Yaskawa INFORM job: test_long_tjr1.JBI

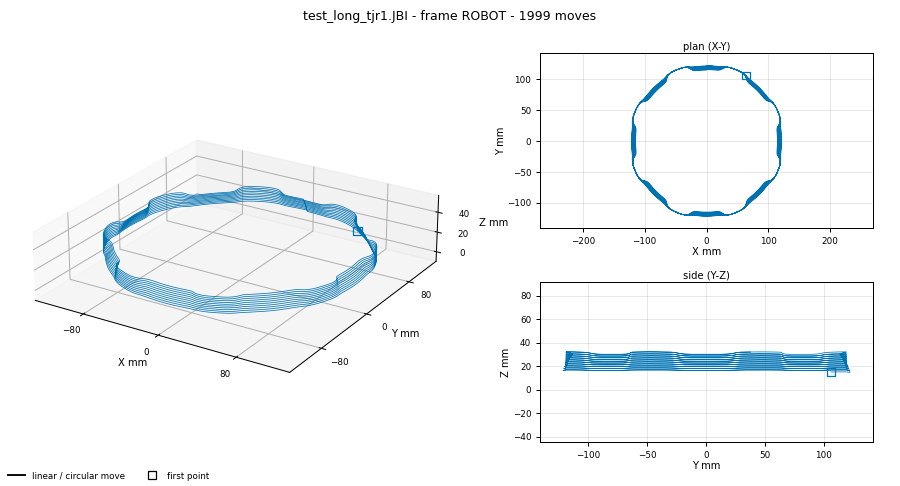
[picture p0: tool path of test_long_tjr1.JBI in frame ROBOT, 1999 of 2000 moves have a stored position in this frame; points joined in program order, loops and branches not executed]
version: 0
/JOB
//NAME test_long
//POS
///NPOS 48,0,0,2,0,0
///TOOL 1
///POSTYPE ROBOT
///RECTAN
///RCONF 1,0,0,0,0,0,0,0,0,0,0,0,0,0,0,0,0,0,0,0,0,0,0,0
C00000=65.650,104.570,15.190,-0.1200,-0.1200,0.9800
C00001=64.100,106.080,15.240,-0.0800,-0.0900,0.9900
C00002=62.010,107.790,15.260,-0.0400,-0.0600,1.0000
C00003=59.150,109.770,15.270,-0.0200,-0.0300,1.0000
C00004=55.850,111.730,15.280,-0.0000,-0.0100,1.0000
C00005=52.540,113.410,15.290,-0.0000,-0.0000,1.0000
C00006=49.390,114.830,15.300,-0.0000,-0.0000,1.0000
C00007=46.270,116.120,15.300,-0.0000,-0.0000,1.0000
C00008=43.040,117.340,15.290,-0.0000,-0.0000,1.0000
C00009=39.510,118.500,15.280,-0.0000,-0.0100,1.0000
C00010=35.790,119.440,15.270,-0.0100,-0.0300,1.0000
C00011=32.370,120.070,15.260,-0.0100,-0.0700,1.0000
C00012=29.680,120.330,15.240,-0.0100,-0.1200,0.9900
C00013=27.520,120.360,15.190,0.0000,-0.1700,0.9800
C00014=25.390,120.360,15.130,-0.0000,-0.2300,0.9700
C00015=22.760,120.490,15.060,-0.0200,-0.2800,0.9600
C00016=18.940,120.890,15.000,-0.0400,-0.3200,0.9500
C00017=13.310,121.540,14.980,-0.0300,-0.3300,0.9400
C00018=6.990,122.060,14.980,-0.0200,-0.3300,0.9400
C00019=0.000,122.260,14.980,0.0000,-0.3300,0.9400
C00020=0.000,121.680,16.580,0.0000,-0.3600,0.9300
C00021=6.940,121.480,16.570,-0.0200,-0.3600,0.9300
C00022=13.220,120.960,16.580,-0.0400,-0.3500,0.9300
C00023=18.830,120.330,16.610,-0.0400,-0.3400,0.9400
C00024=22.630,119.990,16.680,-0.0100,-0.3100,0.9500
C00025=25.240,119.950,16.770,0.0100,-0.2500,0.9700
C00026=27.360,120.050,16.860,0.0100,-0.1800,0.9800
C00027=29.510,120.140,16.920,0.0000,-0.1200,0.9900
C00028=32.190,119.970,16.950,-0.0100,-0.0700,1.0000
C00029=35.620,119.420,16.970,-0.0100,-0.0300,1.0000
C00030=39.380,118.520,16.980,-0.0000,-0.0100,1.0000
C00031=42.960,117.370,16.990,-0.0000,-0.0000,1.0000
C00032=46.240,116.130,17.000,-0.0000,-0.0000,1.0000
C00033=49.420,114.820,17.000,-0.0000,-0.0000,1.0000
C00034=52.620,113.370,16.990,-0.0000,-0.0000,1.0000
C00035=55.960,111.650,16.980,-0.0000,-0.0100,1.0000
C00036=59.250,109.630,16.970,-0.0200,-0.0300,1.0000
C00037=62.070,107.590,16.950,-0.0500,-0.0600,1.0000
C00038=64.080,105.820,16.920,-0.0900,-0.0900,0.9900
C00039=65.540,104.240,16.860,-0.1400,-0.1200,0.9800
C00040=66.970,102.660,16.770,-0.1800,-0.1700,0.9700
C00041=68.850,100.850,16.680,-0.2100,-0.2300,0.9500
C00042=71.770,98.410,16.610,-0.2200,-0.2700,0.9400
C00043=76.180,94.880,16.580,-0.2300,-0.2800,0.9300
C00044=80.990,90.800,16.570,-0.2400,-0.2700,0.9300
C00045=86.040,86.040,16.580,-0.2500,-0.2500,0.9300
C00046=90.800,80.990,16.570,-0.2700,-0.2400,0.9300
C00047=94.880,76.180,16.580,-0.2800,-0.2300,0.9300
C00048=98.410,71.770,16.610,-0.2700,-0.2200,0.9400
C00049=100.850,68.850,16.680,-0.2300,-0.2100,0.9500
C00050=102.660,66.970,16.770,-0.1700,-0.1800,0.9700
C00051=104.240,65.540,16.860,-0.1200,-0.1400,0.9800
C00052=105.820,64.080,16.920,-0.0900,-0.0900,0.9900
C00053=107.590,62.070,16.950,-0.0600,-0.0500,1.0000
C00054=109.630,59.250,16.970,-0.0300,-0.0200,1.0000
C00055=111.650,55.960,16.980,-0.0100,-0.0000,1.0000
C00056=113.370,52.620,16.990,-0.0000,-0.0000,1.0000
C00057=114.820,49.420,17.000,-0.0000,-0.0000,1.0000
C00058=116.130,46.240,17.000,-0.0000,-0.0000,1.0000
C00059=117.370,42.960,16.990,-0.0000,-0.0000,1.0000
C00060=118.520,39.380,16.980,-0.0100,-0.0000,1.0000
C00061=119.420,35.620,16.970,-0.0300,-0.0100,1.0000
C00062=119.970,32.190,16.950,-0.0700,-0.0100,1.0000
C00063=120.140,29.510,16.920,-0.1200,0.0000,0.9900
C00064=120.050,27.360,16.860,-0.1800,0.0100,0.9800
C00065=119.950,25.240,16.770,-0.2500,0.0100,0.9700
C00066=119.990,22.630,16.680,-0.3100,-0.0100,0.9500
C00067=120.330,18.830,16.610,-0.3400,-0.0400,0.9400
C00068=120.960,13.220,16.580,-0.3500,-0.0400,0.9300
C00069=121.480,6.940,16.570,-0.3600,-0.0200,0.9300
C00070=121.680,0.000,16.580,-0.3600,0.0000,0.9300
C00071=121.480,-6.940,16.570,-0.3600,0.0200,0.9300
C00072=120.960,-13.220,16.580,-0.3500,0.0400,0.9300
C00073=120.330,-18.830,16.610,-0.3400,0.0400,0.9400
C00074=119.990,-22.630,16.680,-0.3100,0.0100,0.9500
C00075=119.950,-25.240,16.770,-0.2500,-0.0100,0.9700
C00076=120.050,-27.360,16.860,-0.1800,-0.0100,0.9800
C00077=120.140,-29.510,16.920,-0.1200,-0.0000,0.9900
C00078=119.970,-32.190,16.950,-0.0700,0.0100,1.0000
C00079=119.420,-35.620,16.970,-0.0300,0.0100,1.0000
C00080=118.520,-39.380,16.980,-0.0100,0.0000,1.0000
C00081=117.370,-42.960,16.990,-0.0000,0.0000,1.0000
C00082=116.130,-46.240,17.000,-0.0000,0.0000,1.0000
C00083=114.820,-49.420,17.000,-0.0000,0.0000,1.0000
C00084=113.370,-52.620,16.990,-0.0000,0.0000,1.0000
C00085=111.650,-55.960,16.980,-0.0100,0.0000,1.0000
C00086=109.630,-59.250,16.970,-0.0300,0.0200,1.0000
C00087=107.590,-62.070,16.950,-0.0600,0.0500,1.0000
C00088=105.820,-64.080,16.920,-0.0900,0.0900,0.9900
C00089=104.240,-65.540,16.860,-0.1200,0.1400,0.9800
C00090=102.660,-66.970,16.770,-0.1700,0.1800,0.9700
C00091=100.850,-68.850,16.680,-0.2300,0.2100,0.9500
C00092=98.410,-71.770,16.610,-0.2700,0.2200,0.9400
C00093=94.880,-76.180,16.580,-0.2800,0.2300,0.9300
C00094=90.800,-80.990,16.570,-0.2700,0.2400,0.9300
C00095=86.040,-86.040,16.580,-0.2500,0.2500,0.9300
C00096=80.990,-90.800,16.570,-0.2400,0.2700,0.9300
C00097=76.180,-94.880,16.580,-0.2300,0.2800,0.9300
C00098=71.770,-98.410,16.610,-0.2200,0.2700,0.9400
C00099=68.850,-100.850,16.680,-0.2100,0.2300,0.9500
C00100=66.970,-102.660,16.770,-0.1800,0.1700,0.9700
C00101=65.540,-104.240,16.860,-0.1400,0.1200,0.9800
C00102=64.080,-105.820,16.920,-0.0900,0.0900,0.9900
C00103=62.070,-107.590,16.950,-0.0500,0.0600,1.0000
C00104=59.250,-109.630,16.970,-0.0200,0.0300,1.0000
C00105=55.960,-111.650,16.980,-0.0000,0.0100,1.0000
C00106=52.620,-113.370,16.990,-0.0000,0.0000,1.0000
C00107=49.420,-114.820,17.000,-0.0000,0.0000,1.0000
C00108=46.240,-116.130,17.000,-0.0000,0.0000,1.0000
C00109=42.960,-117.370,16.990,-0.0000,0.0000,1.0000
C00110=39.380,-118.520,16.980,-0.0000,0.0100,1.0000
C00111=35.620,-119.420,16.970,-0.0100,0.0300,1.0000
C00112=32.190,-119.970,16.950,-0.0100,0.0700,1.0000
C00113=29.510,-120.140,16.920,0.0000,0.1200,0.9900
C00114=27.360,-120.050,16.860,0.0100,0.1800,0.9800
C00115=25.240,-119.950,16.770,0.0100,0.2500,0.9700
C00116=22.630,-119.990,16.680,-0.0100,0.3100,0.9500
C00117=18.830,-120.330,16.610,-0.0400,0.3400,0.9400
C00118=13.220,-120.960,16.580,-0.0400,0.3500,0.9300
C00119=6.940,-121.480,16.570,-0.0200,0.3600,0.9300
C00120=0.000,-121.680,16.580,0.0000,0.3600,0.9300
C00121=0.000,-121.680,16.580,0.0000,0.3600,0.9300
C00122=-6.940,-121.480,16.570,0.0200,0.3600,0.9300
C00123=-13.220,-120.960,16.580,0.0400,0.3500,0.9300
C00124=-18.830,-120.330,16.610,0.0400,0.3400,0.9400
C00125=-22.630,-119.990,16.680,0.0100,0.3100,0.9500
C00126=-25.240,-119.950,16.770,-0.0100,0.2500,0.9700
C00127=-27.360,-120.050,16.860,-0.0100,0.1800,0.9800
C00128=-29.510,-120.140,16.920,-0.0000,0.1200,0.9900
C00129=-32.190,-119.970,16.950,0.0100,0.0700,1.0000
C00130=-35.620,-119.420,16.970,0.0100,0.0300,1.0000
C00131=-39.380,-118.520,16.980,0.0000,0.0100,1.0000
C00132=-42.960,-117.370,16.990,0.0000,0.0000,1.0000
C00133=-46.240,-116.130,17.000,0.0000,0.0000,1.0000
C00134=-49.420,-114.820,17.000,0.0000,0.0000,1.0000
C00135=-52.620,-113.370,16.990,0.0000,0.0000,1.0000
C00136=-55.960,-111.650,16.980,0.0000,0.0100,1.0000
C00137=-59.250,-109.630,16.970,0.0200,0.0300,1.0000
C00138=-62.070,-107.590,16.950,0.0500,0.0600,1.0000
C00139=-64.080,-105.820,16.920,0.0900,0.0900,0.9900
C00140=-65.540,-104.240,16.860,0.1400,0.1200,0.9800
C00141=-66.970,-102.660,16.770,0.1800,0.1700,0.9700
C00142=-68.850,-100.850,16.680,0.2100,0.2300,0.9500
C00143=-71.770,-98.410,16.610,0.2200,0.2700,0.9400
C00144=-76.180,-94.880,16.580,0.2300,0.2800,0.9300
C00145=-80.990,-90.800,16.570,0.2400,0.2700,0.9300
C00146=-86.040,-86.040,16.580,0.2500,0.2500,0.9300
C00147=-90.800,-80.990,16.570,0.2700,0.2400,0.9300
C00148=-94.880,-76.180,16.580,0.2800,0.2300,0.9300
C00149=-98.410,-71.770,16.610,0.2700,0.2200,0.9400
C00150=-100.850,-68.850,16.680,0.2300,0.2100,0.9500
C00151=-102.660,-66.970,16.770,0.1700,0.1800,0.9700
C00152=-104.240,-65.540,16.860,0.1200,0.1400,0.9800
C00153=-105.820,-64.080,16.920,0.0900,0.0900,0.9900
C00154=-107.590,-62.070,16.950,0.0600,0.0500,1.0000
C00155=-109.630,-59.250,16.970,0.0300,0.0200,1.0000
C00156=-111.650,-55.960,16.980,0.0100,0.0000,1.0000
C00157=-113.370,-52.620,16.990,0.0000,0.0000,1.0000
C00158=-114.820,-49.420,17.000,0.0000,0.0000,1.0000
C00159=-116.130,-46.240,17.000,0.0000,0.0000,1.0000
C00160=-117.370,-42.960,16.990,0.0000,0.0000,1.0000
C00161=-118.520,-39.380,16.980,0.0100,0.0000,1.0000
C00162=-119.420,-35.620,16.970,0.0300,0.0100,1.0000
C00163=-119.970,-32.190,16.950,0.0700,0.0100,1.0000
C00164=-120.140,-29.510,16.920,0.1200,-0.0000,0.9900
C00165=-120.050,-27.360,16.860,0.1800,-0.0100,0.9800
C00166=-119.950,-25.240,16.770,0.2500,-0.0100,0.9700
C00167=-119.990,-22.630,16.680,0.3100,0.0100,0.9500
C00168=-120.330,-18.830,16.610,0.3400,0.0400,0.9400
C00169=-120.960,-13.220,16.580,0.3500,0.0400,0.9300
C00170=-121.480,-6.940,16.570,0.3600,0.0200,0.9300
C00171=-121.680,0.000,16.580,0.3600,-0.0000,0.9300
C00172=-121.480,6.940,16.570,0.3600,-0.0200,0.9300
C00173=-120.960,13.220,16.580,0.3500,-0.0400,0.9300
C00174=-120.330,18.830,16.610,0.3400,-0.0400,0.9400
C00175=-119.990,22.630,16.680,0.3100,-0.0100,0.9500
C00176=-119.950,25.240,16.770,0.2500,0.0100,0.9700
C00177=-120.050,27.360,16.860,0.1800,0.0100,0.9800
C00178=-120.140,29.510,16.920,0.1200,0.0000,0.9900
C00179=-119.970,32.190,16.950,0.0700,-0.0100,1.0000
C00180=-119.420,35.620,16.970,0.0300,-0.0100,1.0000
C00181=-118.520,39.380,16.980,0.0100,-0.0000,1.0000
C00182=-117.370,42.960,16.990,0.0000,-0.0000,1.0000
C00183=-116.130,46.240,17.000,0.0000,-0.0000,1.0000
C00184=-114.820,49.420,17.000,0.0000,-0.0000,1.0000
C00185=-113.370,52.620,16.990,0.0000,-0.0000,1.0000
C00186=-111.650,55.960,16.980,0.0100,-0.0000,1.0000
C00187=-109.630,59.250,16.970,0.0300,-0.0200,1.0000
C00188=-107.590,62.070,16.950,0.0600,-0.0500,1.0000
C00189=-105.820,64.080,16.920,0.0900,-0.0900,0.9900
C00190=-104.240,65.540,16.860,0.1200,-0.1400,0.9800
C00191=-102.660,66.970,16.770,0.1700,-0.1800,0.9700
C00192=-100.850,68.850,16.680,0.2300,-0.2100,0.9500
C00193=-98.410,71.770,16.610,0.2700,-0.2200,0.9400
C00194=-94.880,76.180,16.580,0.2800,-0.2300,0.9300
C00195=-90.800,80.990,16.570,0.2700,-0.2400,0.9300
C00196=-86.040,86.040,16.580,0.2500,-0.2500,0.9300
C00197=-80.990,90.800,16.570,0.2400,-0.2700,0.9300
C00198=-76.180,94.880,16.580,0.2300,-0.2800,0.9300
C00199=-71.770,98.410,16.610,0.2200,-0.2700,0.9400
C00200=-68.850,100.850,16.680,0.2100,-0.2300,0.9500
C00201=-66.970,102.660,16.770,0.1800,-0.1700,0.9700
C00202=-65.540,104.240,16.860,0.1400,-0.1200,0.9800
C00203=-64.080,105.820,16.920,0.0900,-0.0900,0.9900
C00204=-62.070,107.590,16.950,0.0500,-0.0600,1.0000
C00205=-59.250,109.630,16.970,0.0200,-0.0300,1.0000
C00206=-55.960,111.650,16.980,0.0000,-0.0100,1.0000
C00207=-52.620,113.370,16.990,0.0000,-0.0000,1.0000
C00208=-49.420,114.820,17.000,0.0000,-0.0000,1.0000
C00209=-46.240,116.130,17.000,0.0000,-0.0000,1.0000
C00210=-42.960,117.370,16.990,0.0000,-0.0000,1.0000
C00211=-39.380,118.520,16.980,0.0000,-0.0100,1.0000
C00212=-35.620,119.420,16.970,0.0100,-0.0300,1.0000
C00213=-32.190,119.970,16.950,0.0100,-0.0700,1.0000
C00214=-29.510,120.140,16.920,-0.0000,-0.1200,0.9900
C00215=-27.360,120.050,16.860,-0.0100,-0.1800,0.9800
C00216=-25.240,119.950,16.770,-0.0100,-0.2500,0.9700
C00217=-22.630,119.990,16.680,0.0100,-0.3100,0.9500
C00218=-18.830,120.330,16.610,0.0400,-0.3400,0.9400
C00219=-13.220,120.960,16.580,0.0400,-0.3500,0.9300
C00220=-6.940,121.480,16.570,0.0200,-0.3600,0.9300
C00221=0.000,121.680,16.580,0.0000,-0.3600,0.9300
C00222=0.000,121.050,18.160,0.0000,-0.3800,0.9200
C00223=-6.880,120.850,18.150,0.0200,-0.3800,0.9200
C00224=-13.130,120.340,18.160,0.0400,-0.3800,0.9200
C00225=-18.720,119.740,18.190,0.0400,-0.3700,0.9300
C00226=-22.490,119.460,18.290,0.0100,-0.3300,0.9400
C00227=-25.080,119.500,18.400,-0.0200,-0.2600,0.9600
C00228=-27.190,119.720,18.520,-0.0200,-0.1900,0.9800
C00229=-29.330,119.920,18.600,-0.0100,-0.1300,0.9900
C00230=-31.990,119.860,18.640,0.0100,-0.0700,1.0000
C00231=-35.440,119.400,18.660,0.0100,-0.0300,1.0000
C00232=-39.230,118.550,18.670,0.0000,-0.0100,1.0000
C00233=-42.870,117.400,18.690,0.0000,-0.0000,1.0000
C00234=-46.210,116.140,18.700,0.0000,-0.0000,1.0000
C00235=-49.450,114.800,18.700,0.0000,-0.0000,1.0000
C00236=-52.700,113.320,18.690,0.0000,-0.0000,1.0000
C00237=-56.080,111.570,18.670,0.0000,-0.0100,1.0000
C00238=-59.370,109.490,18.660,0.0200,-0.0300,1.0000
C00239=-62.130,107.380,18.640,0.0500,-0.0600,1.0000
C00240=-64.050,105.540,18.600,0.0900,-0.0800,0.9900
C00241=-65.430,103.880,18.520,0.1500,-0.1200,0.9800
C00242=-66.770,102.230,18.400,0.2000,-0.1700,0.9600
C00243=-68.570,100.370,18.290,0.2300,-0.2400,0.9400
C00244=-71.430,97.900,18.190,0.2300,-0.2800,0.9300
C00245=-75.810,94.380,18.160,0.2400,-0.3000,0.9200
C00246=-80.590,90.320,18.150,0.2500,-0.2900,0.9200
C00247=-85.590,85.590,18.160,0.2700,-0.2700,0.9200
C00248=-90.320,80.590,18.150,0.2900,-0.2500,0.9200
C00249=-94.380,75.810,18.160,0.3000,-0.2400,0.9200
C00250=-97.900,71.430,18.190,0.2800,-0.2300,0.9300
C00251=-100.370,68.570,18.290,0.2400,-0.2300,0.9400
C00252=-102.230,66.770,18.400,0.1700,-0.2000,0.9600
C00253=-103.880,65.430,18.520,0.1200,-0.1500,0.9800
C00254=-105.540,64.050,18.600,0.0800,-0.0900,0.9900
C00255=-107.380,62.130,18.640,0.0600,-0.0500,1.0000
C00256=-109.490,59.370,18.660,0.0300,-0.0200,1.0000
C00257=-111.570,56.080,18.670,0.0100,-0.0000,1.0000
C00258=-113.320,52.700,18.690,0.0000,-0.0000,1.0000
C00259=-114.800,49.450,18.700,0.0000,-0.0000,1.0000
C00260=-116.140,46.210,18.700,0.0000,-0.0000,1.0000
C00261=-117.400,42.870,18.690,0.0000,-0.0000,1.0000
C00262=-118.550,39.230,18.670,0.0100,-0.0000,1.0000
C00263=-119.400,35.440,18.660,0.0300,-0.0100,1.0000
C00264=-119.860,31.990,18.640,0.0700,-0.0100,1.0000
C00265=-119.920,29.330,18.600,0.1300,0.0100,0.9900
C00266=-119.720,27.190,18.520,0.1900,0.0200,0.9800
C00267=-119.500,25.080,18.400,0.2600,0.0200,0.9600
C00268=-119.460,22.490,18.290,0.3300,-0.0100,0.9400
C00269=-119.740,18.720,18.190,0.3700,-0.0400,0.9300
C00270=-120.340,13.130,18.160,0.3800,-0.0400,0.9200
C00271=-120.850,6.880,18.150,0.3800,-0.0200,0.9200
C00272=-121.050,0.000,18.160,0.3800,-0.0000,0.9200
C00273=-120.850,-6.880,18.150,0.3800,0.0200,0.9200
C00274=-120.340,-13.130,18.160,0.3800,0.0400,0.9200
C00275=-119.740,-18.720,18.190,0.3700,0.0400,0.9300
C00276=-119.460,-22.490,18.290,0.3300,0.0100,0.9400
C00277=-119.500,-25.080,18.400,0.2600,-0.0200,0.9600
C00278=-119.720,-27.190,18.520,0.1900,-0.0200,0.9800
C00279=-119.920,-29.330,18.600,0.1300,-0.0100,0.9900
C00280=-119.860,-31.990,18.640,0.0700,0.0100,1.0000
C00281=-119.400,-35.440,18.660,0.0300,0.0100,1.0000
C00282=-118.550,-39.230,18.670,0.0100,0.0000,1.0000
C00283=-117.400,-42.870,18.690,0.0000,0.0000,1.0000
C00284=-116.140,-46.210,18.700,0.0000,0.0000,1.0000
C00285=-114.800,-49.450,18.700,0.0000,0.0000,1.0000
C00286=-113.320,-52.700,18.690,0.0000,0.0000,1.0000
C00287=-111.570,-56.080,18.670,0.0100,0.0000,1.0000
C00288=-109.490,-59.370,18.660,0.0300,0.0200,1.0000
C00289=-107.380,-62.130,18.640,0.0600,0.0500,1.0000
C00290=-105.540,-64.050,18.600,0.0800,0.0900,0.9900
C00291=-103.880,-65.430,18.520,0.1200,0.1500,0.9800
C00292=-102.230,-66.770,18.400,0.1700,0.2000,0.9600
C00293=-100.370,-68.570,18.290,0.2400,0.2300,0.9400
C00294=-97.900,-71.430,18.190,0.2800,0.2300,0.9300
C00295=-94.380,-75.810,18.160,0.3000,0.2400,0.9200
C00296=-90.320,-80.590,18.150,0.2900,0.2500,0.9200
C00297=-85.590,-85.590,18.160,0.2700,0.2700,0.9200
C00298=-80.590,-90.320,18.150,0.2500,0.2900,0.9200
C00299=-75.810,-94.380,18.160,0.2400,0.3000,0.9200
C00300=-71.430,-97.900,18.190,0.2300,0.2800,0.9300
C00301=-68.570,-100.370,18.290,0.2300,0.2400,0.9400
C00302=-66.770,-102.230,18.400,0.2000,0.1700,0.9600
C00303=-65.430,-103.880,18.520,0.1500,0.1200,0.9800
C00304=-64.050,-105.540,18.600,0.0900,0.0800,0.9900
C00305=-62.130,-107.380,18.640,0.0500,0.0600,1.0000
C00306=-59.370,-109.490,18.660,0.0200,0.0300,1.0000
C00307=-56.080,-111.570,18.670,0.0000,0.0100,1.0000
C00308=-52.700,-113.320,18.690,0.0000,0.0000,1.0000
C00309=-49.450,-114.800,18.700,0.0000,0.0000,1.0000
C00310=-46.210,-116.140,18.700,0.0000,0.0000,1.0000
C00311=-42.870,-117.400,18.690,0.0000,0.0000,1.0000
C00312=-39.230,-118.550,18.670,0.0000,0.0100,1.0000
C00313=-35.440,-119.400,18.660,0.0100,0.0300,1.0000
C00314=-31.990,-119.860,18.640,0.0100,0.0700,1.0000
C00315=-29.330,-119.920,18.600,-0.0100,0.1300,0.9900
C00316=-27.190,-119.720,18.520,-0.0200,0.1900,0.9800
C00317=-25.080,-119.500,18.400,-0.0200,0.2600,0.9600
C00318=-22.490,-119.460,18.290,0.0100,0.3300,0.9400
C00319=-18.720,-119.740,18.190,0.0400,0.3700,0.9300
C00320=-13.130,-120.340,18.160,0.0400,0.3800,0.9200
C00321=-6.880,-120.850,18.150,0.0200,0.3800,0.9200
C00322=0.000,-121.050,18.160,0.0000,0.3800,0.9200
C00323=0.000,-121.050,18.160,0.0000,0.3800,0.9200
C00324=6.880,-120.850,18.150,-0.0200,0.3800,0.9200
C00325=13.130,-120.340,18.160,-0.0400,0.3800,0.9200
C00326=18.720,-119.740,18.190,-0.0400,0.3700,0.9300
C00327=22.490,-119.460,18.290,-0.0100,0.3300,0.9400
C00328=25.080,-119.500,18.400,0.0200,0.2600,0.9600
C00329=27.190,-119.720,18.520,0.0200,0.1900,0.9800
C00330=29.330,-119.920,18.600,0.0100,0.1300,0.9900
C00331=31.990,-119.860,18.640,-0.0100,0.0700,1.0000
C00332=35.440,-119.400,18.660,-0.0100,0.0300,1.0000
C00333=39.230,-118.550,18.670,-0.0000,0.0100,1.0000
C00334=42.870,-117.400,18.690,-0.0000,0.0000,1.0000
C00335=46.210,-116.140,18.700,-0.0000,0.0000,1.0000
C00336=49.450,-114.800,18.700,-0.0000,0.0000,1.0000
C00337=52.700,-113.320,18.690,-0.0000,0.0000,1.0000
C00338=56.080,-111.570,18.670,-0.0000,0.0100,1.0000
C00339=59.370,-109.490,18.660,-0.0200,0.0300,1.0000
C00340=62.130,-107.380,18.640,-0.0500,0.0600,1.0000
C00341=64.050,-105.540,18.600,-0.0900,0.0800,0.9900
C00342=65.430,-103.880,18.520,-0.1500,0.1200,0.9800
C00343=66.770,-102.230,18.400,-0.2000,0.1700,0.9600
C00344=68.570,-100.370,18.290,-0.2300,0.2400,0.9400
C00345=71.430,-97.900,18.190,-0.2300,0.2800,0.9300
C00346=75.810,-94.380,18.160,-0.2400,0.3000,0.9200
C00347=80.590,-90.320,18.150,-0.2500,0.2900,0.9200
C00348=85.590,-85.590,18.160,-0.2700,0.2700,0.9200
C00349=90.320,-80.590,18.150,-0.2900,0.2500,0.9200
C00350=94.380,-75.810,18.160,-0.3000,0.2400,0.9200
C00351=97.900,-71.430,18.190,-0.2800,0.2300,0.9300
C00352=100.370,-68.570,18.290,-0.2400,0.2300,0.9400
C00353=102.230,-66.770,18.400,-0.1700,0.2000,0.9600
C00354=103.880,-65.430,18.520,-0.1200,0.1500,0.9800
C00355=105.540,-64.050,18.600,-0.0800,0.0900,0.9900
C00356=107.380,-62.130,18.640,-0.0600,0.0500,1.0000
C00357=109.490,-59.370,18.660,-0.0300,0.0200,1.0000
C00358=111.570,-56.080,18.670,-0.0100,0.0000,1.0000
C00359=113.320,-52.700,18.690,-0.0000,0.0000,1.0000
C00360=114.800,-49.450,18.700,-0.0000,0.0000,1.0000
C00361=116.140,-46.210,18.700,-0.0000,0.0000,1.0000
C00362=117.400,-42.870,18.690,-0.0000,0.0000,1.0000
C00363=118.550,-39.230,18.670,-0.0100,0.0000,1.0000
C00364=119.400,-35.440,18.660,-0.0300,0.0100,1.0000
C00365=119.860,-31.990,18.640,-0.0700,0.0100,1.0000
C00366=119.920,-29.330,18.600,-0.1300,-0.0100,0.9900
C00367=119.720,-27.190,18.520,-0.1900,-0.0200,0.9800
C00368=119.500,-25.080,18.400,-0.2600,-0.0200,0.9600
C00369=119.460,-22.490,18.290,-0.3300,0.0100,0.9400
C00370=119.740,-18.720,18.190,-0.3700,0.0400,0.9300
C00371=120.340,-13.130,18.160,-0.3800,0.0400,0.9200
C00372=120.850,-6.880,18.150,-0.3800,0.0200,0.9200
C00373=121.050,0.000,18.160,-0.3800,0.0000,0.9200
C00374=120.850,6.880,18.150,-0.3800,-0.0200,0.9200
C00375=120.340,13.130,18.160,-0.3800,-0.0400,0.9200
C00376=119.740,18.720,18.190,-0.3700,-0.0400,0.9300
C00377=119.460,22.490,18.290,-0.3300,-0.0100,0.9400
C00378=119.500,25.080,18.400,-0.2600,0.0200,0.9600
C00379=119.720,27.190,18.520,-0.1900,0.0200,0.9800
C00380=119.920,29.330,18.600,-0.1300,0.0100,0.9900
C00381=119.860,31.990,18.640,-0.0700,-0.0100,1.0000
C00382=119.400,35.440,18.660,-0.0300,-0.0100,1.0000
C00383=118.550,39.230,18.670,-0.0100,-0.0000,1.0000
C00384=117.400,42.870,18.690,-0.0000,-0.0000,1.0000
C00385=116.140,46.210,18.700,-0.0000,-0.0000,1.0000
C00386=114.800,49.450,18.700,-0.0000,-0.0000,1.0000
C00387=113.320,52.700,18.690,-0.0000,-0.0000,1.0000
C00388=111.570,56.080,18.670,-0.0100,-0.0000,1.0000
C00389=109.490,59.370,18.660,-0.0300,-0.0200,1.0000
C00390=107.380,62.130,18.640,-0.0600,-0.0500,1.0000
C00391=105.540,64.050,18.600,-0.0800,-0.0900,0.9900
C00392=103.880,65.430,18.520,-0.1200,-0.1500,0.9800
C00393=102.230,66.770,18.400,-0.1700,-0.2000,0.9600
C00394=100.370,68.570,18.290,-0.2400,-0.2300,0.9400
C00395=97.900,71.430,18.190,-0.2800,-0.2300,0.9300
C00396=94.380,75.810,18.160,-0.3000,-0.2400,0.9200
C00397=90.320,80.590,18.150,-0.2900,-0.2500,0.9200
C00398=85.590,85.590,18.160,-0.2700,-0.2700,0.9200
C00399=80.590,90.320,18.150,-0.2500,-0.2900,0.9200
C00400=75.810,94.380,18.160,-0.2400,-0.3000,0.9200
C00401=71.430,97.900,18.190,-0.2300,-0.2800,0.9300
C00402=68.570,100.370,18.290,-0.2300,-0.2400,0.9400
C00403=66.770,102.230,18.400,-0.2000,-0.1700,0.9600
C00404=65.430,103.880,18.520,-0.1500,-0.1200,0.9800
C00405=64.050,105.540,18.600,-0.0900,-0.0800,0.9900
C00406=62.130,107.380,18.640,-0.0500,-0.0600,1.0000
C00407=59.370,109.490,18.660,-0.0200,-0.0300,1.0000
C00408=56.080,111.570,18.670,-0.0000,-0.0100,1.0000
C00409=52.700,113.320,18.690,-0.0000,-0.0000,1.0000
C00410=49.450,114.800,18.700,-0.0000,-0.0000,1.0000
C00411=46.210,116.140,18.700,-0.0000,-0.0000,1.0000
C00412=42.870,117.400,18.690,-0.0000,-0.0000,1.0000
C00413=39.230,118.550,18.670,-0.0000,-0.0100,1.0000
C00414=35.440,119.400,18.660,-0.0100,-0.0300,1.0000
C00415=31.990,119.860,18.640,-0.0100,-0.0700,1.0000
C00416=29.330,119.920,18.600,0.0100,-0.1300,0.9900
C00417=27.190,119.720,18.520,0.0200,-0.1900,0.9800
C00418=25.080,119.500,18.400,0.0200,-0.2600,0.9600
C00419=22.490,119.460,18.290,-0.0100,-0.3300,0.9400
C00420=18.720,119.740,18.190,-0.0400,-0.3700,0.9300
C00421=13.130,120.340,18.160,-0.0400,-0.3800,0.9200
C00422=6.880,120.850,18.150,-0.0200,-0.3800,0.9200
C00423=0.000,121.050,18.160,0.0000,-0.3800,0.9200
C00424=0.000,120.380,19.720,0.0000,-0.4000,0.9100
C00425=6.820,120.180,19.720,-0.0200,-0.4000,0.9100
C00426=13.030,119.680,19.720,-0.0400,-0.4000,0.9100
C00427=18.590,119.100,19.770,-0.0300,-0.3900,0.9200
C00428=22.340,118.890,19.880,0.0000,-0.3500,0.9400
C00429=24.910,119.030,20.030,0.0400,-0.2700,0.9600
C00430=27.010,119.360,20.170,0.0400,-0.1900,0.9800
C00431=29.140,119.690,20.270,0.0100,-0.1300,0.9900
C00432=31.780,119.750,20.320,-0.0000,-0.0800,1.0000
C00433=35.240,119.380,20.340,-0.0100,-0.0300,1.0000
C00434=39.080,118.580,20.360,-0.0000,-0.0100,1.0000
C00435=42.770,117.430,20.380,-0.0000,-0.0000,1.0000
C00436=46.180,116.150,20.400,-0.0000,-0.0000,1.0000
C00437=49.480,114.790,20.400,-0.0000,-0.0000,1.0000
C00438=52.800,113.280,20.380,-0.0000,-0.0000,1.0000
C00439=56.220,111.480,20.360,-0.0000,-0.0100,1.0000
C00440=59.490,109.330,20.340,-0.0200,-0.0300,1.0000
C00441=62.200,107.150,20.320,-0.0500,-0.0600,1.0000
C00442=64.030,105.240,20.270,-0.1000,-0.0800,0.9900
C00443=65.300,103.500,20.170,-0.1600,-0.1100,0.9800
C00444=66.550,101.780,20.030,-0.2200,-0.1700,0.9600
C00445=68.270,99.860,19.880,-0.2500,-0.2400,0.9400
C00446=71.070,97.360,19.770,-0.2500,-0.3000,0.9200
C00447=75.420,93.840,19.720,-0.2600,-0.3100,0.9100
C00448=80.160,89.800,19.720,-0.2700,-0.3000,0.9100
C00449=85.120,85.120,19.720,-0.2900,-0.2900,0.9100
C00450=89.800,80.160,19.720,-0.3000,-0.2700,0.9100
C00451=93.840,75.420,19.720,-0.3100,-0.2600,0.9100
C00452=97.360,71.070,19.770,-0.3000,-0.2500,0.9200
C00453=99.860,68.270,19.880,-0.2400,-0.2500,0.9400
C00454=101.780,66.550,20.030,-0.1700,-0.2200,0.9600
C00455=103.500,65.300,20.170,-0.1100,-0.1600,0.9800
C00456=105.240,64.030,20.270,-0.0800,-0.1000,0.9900
C00457=107.150,62.200,20.320,-0.0600,-0.0500,1.0000
C00458=109.330,59.490,20.340,-0.0300,-0.0200,1.0000
C00459=111.480,56.220,20.360,-0.0100,-0.0000,1.0000
C00460=113.280,52.800,20.380,-0.0000,-0.0000,1.0000
C00461=114.790,49.480,20.400,-0.0000,-0.0000,1.0000
C00462=116.150,46.180,20.400,-0.0000,-0.0000,1.0000
C00463=117.430,42.770,20.380,-0.0000,-0.0000,1.0000
C00464=118.580,39.080,20.360,-0.0100,-0.0000,1.0000
C00465=119.380,35.240,20.340,-0.0300,-0.0100,1.0000
C00466=119.750,31.780,20.320,-0.0800,-0.0000,1.0000
C00467=119.690,29.140,20.270,-0.1300,0.0100,0.9900
C00468=119.360,27.010,20.170,-0.1900,0.0400,0.9800
C00469=119.030,24.910,20.030,-0.2700,0.0400,0.9600
C00470=118.890,22.340,19.880,-0.3500,0.0000,0.9400
C00471=119.100,18.590,19.770,-0.3900,-0.0300,0.9200
C00472=119.680,13.030,19.720,-0.4000,-0.0400,0.9100
C00473=120.180,6.820,19.720,-0.4000,-0.0200,0.9100
C00474=120.380,0.000,19.720,-0.4000,0.0000,0.9100
C00475=120.180,-6.820,19.720,-0.4000,0.0200,0.9100
C00476=119.680,-13.030,19.720,-0.4000,0.0400,0.9100
C00477=119.100,-18.590,19.770,-0.3900,0.0300,0.9200
C00478=118.890,-22.340,19.880,-0.3500,-0.0000,0.9400
C00479=119.030,-24.910,20.030,-0.2700,-0.0400,0.9600
C00480=119.360,-27.010,20.170,-0.1900,-0.0400,0.9800
C00481=119.690,-29.140,20.270,-0.1300,-0.0100,0.9900
C00482=119.750,-31.780,20.320,-0.0800,0.0000,1.0000
C00483=119.380,-35.240,20.340,-0.0300,0.0100,1.0000
C00484=118.580,-39.080,20.360,-0.0100,0.0000,1.0000
C00485=117.430,-42.770,20.380,-0.0000,0.0000,1.0000
C00486=116.150,-46.180,20.400,-0.0000,0.0000,1.0000
C00487=114.790,-49.480,20.400,-0.0000,0.0000,1.0000
C00488=113.280,-52.800,20.380,-0.0000,0.0000,1.0000
C00489=111.480,-56.220,20.360,-0.0100,0.0000,1.0000
C00490=109.330,-59.490,20.340,-0.0300,0.0200,1.0000
C00491=107.150,-62.200,20.320,-0.0600,0.0500,1.0000
C00492=105.240,-64.030,20.270,-0.0800,0.1000,0.9900
C00493=103.500,-65.300,20.170,-0.1100,0.1600,0.9800
C00494=101.780,-66.550,20.030,-0.1700,0.2200,0.9600
C00495=99.860,-68.270,19.880,-0.2400,0.2500,0.9400
C00496=97.360,-71.070,19.770,-0.3000,0.2500,0.9200
C00497=93.840,-75.420,19.720,-0.3100,0.2600,0.9100
C00498=89.800,-80.160,19.720,-0.3000,0.2700,0.9100
C00499=85.120,-85.120,19.720,-0.2900,0.2900,0.9100
C00500=80.160,-89.800,19.720,-0.2700,0.3000,0.9100
C00501=75.420,-93.840,19.720,-0.2600,0.3100,0.9100
C00502=71.070,-97.360,19.770,-0.2500,0.3000,0.9200
C00503=68.270,-99.860,19.880,-0.2500,0.2400,0.9400
C00504=66.550,-101.780,20.030,-0.2200,0.1700,0.9600
C00505=65.300,-103.500,20.170,-0.1600,0.1100,0.9800
C00506=64.030,-105.240,20.270,-0.1000,0.0800,0.9900
C00507=62.200,-107.150,20.320,-0.0500,0.0600,1.0000
C00508=59.490,-109.330,20.340,-0.0200,0.0300,1.0000
C00509=56.220,-111.480,20.360,-0.0000,0.0100,1.0000
C00510=52.800,-113.280,20.380,-0.0000,0.0000,1.0000
C00511=49.480,-114.790,20.400,-0.0000,0.0000,1.0000
C00512=46.180,-116.150,20.400,-0.0000,0.0000,1.0000
C00513=42.770,-117.430,20.380,-0.0000,0.0000,1.0000
C00514=39.080,-118.580,20.360,-0.0000,0.0100,1.0000
C00515=35.240,-119.380,20.340,-0.0100,0.0300,1.0000
C00516=31.780,-119.750,20.320,-0.0000,0.0800,1.0000
C00517=29.140,-119.690,20.270,0.0100,0.1300,0.9900
C00518=27.010,-119.360,20.170,0.0400,0.1900,0.9800
C00519=24.910,-119.030,20.030,0.0400,0.2700,0.9600
C00520=22.340,-118.890,19.880,0.0000,0.3500,0.9400
C00521=18.590,-119.100,19.770,-0.0300,0.3900,0.9200
C00522=13.030,-119.680,19.720,-0.0400,0.4000,0.9100
C00523=6.820,-120.180,19.720,-0.0200,0.4000,0.9100
C00524=0.000,-120.380,19.720,0.0000,0.4000,0.9100
C00525=0.000,-120.380,19.720,0.0000,0.4000,0.9100
C00526=-6.820,-120.180,19.720,0.0200,0.4000,0.9100
C00527=-13.030,-119.680,19.720,0.0400,0.4000,0.9100
C00528=-18.590,-119.100,19.770,0.0300,0.3900,0.9200
C00529=-22.340,-118.890,19.880,-0.0000,0.3500,0.9400
C00530=-24.910,-119.030,20.030,-0.0400,0.2700,0.9600
C00531=-27.010,-119.360,20.170,-0.0400,0.1900,0.9800
C00532=-29.140,-119.690,20.270,-0.0100,0.1300,0.9900
C00533=-31.780,-119.750,20.320,0.0000,0.0800,1.0000
C00534=-35.240,-119.380,20.340,0.0100,0.0300,1.0000
C00535=-39.080,-118.580,20.360,0.0000,0.0100,1.0000
C00536=-42.770,-117.430,20.380,0.0000,0.0000,1.0000
C00537=-46.180,-116.150,20.400,0.0000,0.0000,1.0000
C00538=-49.480,-114.790,20.400,0.0000,0.0000,1.0000
C00539=-52.800,-113.280,20.380,0.0000,0.0000,1.0000
C00540=-56.220,-111.480,20.360,0.0000,0.0100,1.0000
C00541=-59.490,-109.330,20.340,0.0200,0.0300,1.0000
C00542=-62.200,-107.150,20.320,0.0500,0.0600,1.0000
C00543=-64.030,-105.240,20.270,0.1000,0.0800,0.9900
C00544=-65.300,-103.500,20.170,0.1600,0.1100,0.9800
C00545=-66.550,-101.780,20.030,0.2200,0.1700,0.9600
C00546=-68.270,-99.860,19.880,0.2500,0.2400,0.9400
C00547=-71.070,-97.360,19.770,0.2500,0.3000,0.9200
C00548=-75.420,-93.840,19.720,0.2600,0.3100,0.9100
C00549=-80.160,-89.800,19.720,0.2700,0.3000,0.9100
C00550=-85.120,-85.120,19.720,0.2900,0.2900,0.9100
C00551=-89.800,-80.160,19.720,0.3000,0.2700,0.9100
C00552=-93.840,-75.420,19.720,0.3100,0.2600,0.9100
C00553=-97.360,-71.070,19.770,0.3000,0.2500,0.9200
C00554=-99.860,-68.270,19.880,0.2400,0.2500,0.9400
C00555=-101.780,-66.550,20.030,0.1700,0.2200,0.9600
C00556=-103.500,-65.300,20.170,0.1100,0.1600,0.9800
C00557=-105.240,-64.030,20.270,0.0800,0.1000,0.9900
C00558=-107.150,-62.200,20.320,0.0600,0.0500,1.0000
C00559=-109.330,-59.490,20.340,0.0300,0.0200,1.0000
C00560=-111.480,-56.220,20.360,0.0100,0.0000,1.0000
C00561=-113.280,-52.800,20.380,0.0000,0.0000,1.0000
C00562=-114.790,-49.480,20.400,0.0000,0.0000,1.0000
C00563=-116.150,-46.180,20.400,0.0000,0.0000,1.0000
C00564=-117.430,-42.770,20.380,0.0000,0.0000,1.0000
C00565=-118.580,-39.080,20.360,0.0100,0.0000,1.0000
C00566=-119.380,-35.240,20.340,0.0300,0.0100,1.0000
C00567=-119.750,-31.780,20.320,0.0800,0.0000,1.0000
C00568=-119.690,-29.140,20.270,0.1300,-0.0100,0.9900
C00569=-119.360,-27.010,20.170,0.1900,-0.0400,0.9800
C00570=-119.030,-24.910,20.030,0.2700,-0.0400,0.9600
C00571=-118.890,-22.340,19.880,0.3500,-0.0000,0.9400
C00572=-119.100,-18.590,19.770,0.3900,0.0300,0.9200
C00573=-119.680,-13.030,19.720,0.4000,0.0400,0.9100
C00574=-120.180,-6.820,19.720,0.4000,0.0200,0.9100
C00575=-120.380,0.000,19.720,0.4000,-0.0000,0.9100
C00576=-120.180,6.820,19.720,0.4000,-0.0200,0.9100
C00577=-119.680,13.030,19.720,0.4000,-0.0400,0.9100
C00578=-119.100,18.590,19.770,0.3900,-0.0300,0.9200
C00579=-118.890,22.340,19.880,0.3500,0.0000,0.9400
C00580=-119.030,24.910,20.030,0.2700,0.0400,0.9600
C00581=-119.360,27.010,20.170,0.1900,0.0400,0.9800
C00582=-119.690,29.140,20.270,0.1300,0.0100,0.9900
C00583=-119.750,31.780,20.320,0.0800,-0.0000,1.0000
C00584=-119.380,35.240,20.340,0.0300,-0.0100,1.0000
C00585=-118.580,39.080,20.360,0.0100,-0.0000,1.0000
C00586=-117.430,42.770,20.380,0.0000,-0.0000,1.0000
C00587=-116.150,46.180,20.400,0.0000,-0.0000,1.0000
C00588=-114.790,49.480,20.400,0.0000,-0.0000,1.0000
C00589=-113.280,52.800,20.380,0.0000,-0.0000,1.0000
C00590=-111.480,56.220,20.360,0.0100,-0.0000,1.0000
C00591=-109.330,59.490,20.340,0.0300,-0.0200,1.0000
C00592=-107.150,62.200,20.320,0.0600,-0.0500,1.0000
C00593=-105.240,64.030,20.270,0.0800,-0.1000,0.9900
C00594=-103.500,65.300,20.170,0.1100,-0.1600,0.9800
C00595=-101.780,66.550,20.030,0.1700,-0.2200,0.9600
C00596=-99.860,68.270,19.880,0.2400,-0.2500,0.9400
C00597=-97.360,71.070,19.770,0.3000,-0.2500,0.9200
C00598=-93.840,75.420,19.720,0.3100,-0.2600,0.9100
C00599=-89.800,80.160,19.720,0.3000,-0.2700,0.9100
C00600=-85.120,85.120,19.720,0.2900,-0.2900,0.9100
C00601=-80.160,89.800,19.720,0.2700,-0.3000,0.9100
C00602=-75.420,93.840,19.720,0.2600,-0.3100,0.9100
C00603=-71.070,97.360,19.770,0.2500,-0.3000,0.9200
C00604=-68.270,99.860,19.880,0.2500,-0.2400,0.9400
C00605=-66.550,101.780,20.030,0.2200,-0.1700,0.9600
C00606=-65.300,103.500,20.170,0.1600,-0.1100,0.9800
C00607=-64.030,105.240,20.270,0.1000,-0.0800,0.9900
C00608=-62.200,107.150,20.320,0.0500,-0.0600,1.0000
C00609=-59.490,109.330,20.340,0.0200,-0.0300,1.0000
C00610=-56.220,111.480,20.360,0.0000,-0.0100,1.0000
C00611=-52.800,113.280,20.380,0.0000,-0.0000,1.0000
C00612=-49.480,114.790,20.400,0.0000,-0.0000,1.0000
C00613=-46.180,116.150,20.400,0.0000,-0.0000,1.0000
C00614=-42.770,117.430,20.380,0.0000,-0.0000,1.0000
C00615=-39.080,118.580,20.360,0.0000,-0.0100,1.0000
C00616=-35.240,119.380,20.340,0.0100,-0.0300,1.0000
C00617=-31.780,119.750,20.320,0.0000,-0.0800,1.0000
C00618=-29.140,119.690,20.270,-0.0100,-0.1300,0.9900
C00619=-27.010,119.360,20.170,-0.0400,-0.1900,0.9800
C00620=-24.910,119.030,20.030,-0.0400,-0.2700,0.9600
C00621=-22.340,118.890,19.880,-0.0000,-0.3500,0.9400
C00622=-18.590,119.100,19.770,0.0300,-0.3900,0.9200
C00623=-13.030,119.680,19.720,0.0400,-0.4000,0.9100
C00624=-6.820,120.180,19.720,0.0200,-0.4000,0.9100
C00625=0.000,120.380,19.720,0.0000,-0.4000,0.9100
C00626=0.000,119.670,21.260,0.0000,-0.4300,0.9000
C00627=-6.750,119.480,21.260,0.0200,-0.4300,0.9000
C00628=-12.920,118.980,21.270,0.0400,-0.4200,0.9100
C00629=-18.460,118.430,21.320,0.0300,-0.4100,0.9100
C00630=-22.180,118.280,21.460,-0.0200,-0.3600,0.9300
C00631=-24.730,118.520,21.640,-0.0500,-0.2800,0.9600
C00632=-26.820,118.980,21.810,-0.0500,-0.1900,0.9800
C00633=-28.930,119.440,21.940,-0.0200,-0.1300,0.9900
C00634=-31.560,119.630,22.000,0.0000,-0.0800,1.0000
C00635=-35.030,119.350,22.030,0.0000,-0.0300,1.0000
C00636=-38.910,118.610,22.060,0.0000,-0.0100,1.0000
C00637=-42.660,117.470,22.080,0.0000,-0.0000,1.0000
C00638=-46.140,116.170,22.100,0.0000,-0.0000,1.0000
C00639=-49.510,114.770,22.100,0.0000,-0.0000,1.0000
C00640=-52.890,113.230,22.080,0.0000,-0.0000,1.0000
C00641=-56.360,111.380,22.060,0.0000,-0.0100,1.0000
C00642=-59.620,109.160,22.030,0.0200,-0.0300,1.0000
C00643=-62.270,106.900,22.000,0.0500,-0.0500,1.0000
C00644=-64.000,104.920,21.940,0.1000,-0.0700,0.9900
C00645=-65.170,103.090,21.810,0.1700,-0.1000,0.9800
C00646=-66.320,101.290,21.640,0.2300,-0.1600,0.9600
C00647=-67.960,99.320,21.460,0.2700,-0.2400,0.9300
C00648=-70.690,96.800,21.320,0.2700,-0.3100,0.9100
C00649=-75.000,93.270,21.270,0.2700,-0.3300,0.9100
C00650=-79.710,89.260,21.260,0.2800,-0.3200,0.9000
C00651=-84.620,84.620,21.260,0.3000,-0.3000,0.9000
C00652=-89.260,79.710,21.260,0.3200,-0.2800,0.9000
C00653=-93.270,75.000,21.270,0.3300,-0.2700,0.9100
C00654=-96.800,70.690,21.320,0.3100,-0.2700,0.9100
C00655=-99.320,67.960,21.460,0.2400,-0.2700,0.9300
C00656=-101.290,66.320,21.640,0.1600,-0.2300,0.9600
C00657=-103.090,65.170,21.810,0.1000,-0.1700,0.9800
C00658=-104.920,64.000,21.940,0.0700,-0.1000,0.9900
C00659=-106.900,62.270,22.000,0.0500,-0.0500,1.0000
C00660=-109.160,59.620,22.030,0.0300,-0.0200,1.0000
C00661=-111.380,56.360,22.060,0.0100,-0.0000,1.0000
C00662=-113.230,52.890,22.080,0.0000,-0.0000,1.0000
C00663=-114.770,49.510,22.100,0.0000,-0.0000,1.0000
C00664=-116.170,46.140,22.100,0.0000,-0.0000,1.0000
C00665=-117.470,42.660,22.080,0.0000,-0.0000,1.0000
C00666=-118.610,38.910,22.060,0.0100,-0.0000,1.0000
C00667=-119.350,35.030,22.030,0.0300,-0.0000,1.0000
C00668=-119.630,31.560,22.000,0.0800,-0.0000,1.0000
C00669=-119.440,28.930,21.940,0.1300,0.0200,0.9900
C00670=-118.980,26.820,21.810,0.1900,0.0500,0.9800
C00671=-118.520,24.730,21.640,0.2800,0.0500,0.9600
C00672=-118.280,22.180,21.460,0.3600,0.0200,0.9300
C00673=-118.430,18.460,21.320,0.4100,-0.0300,0.9100
C00674=-118.980,12.920,21.270,0.4200,-0.0400,0.9100
C00675=-119.480,6.750,21.260,0.4300,-0.0200,0.9000
C00676=-119.670,0.000,21.260,0.4300,-0.0000,0.9000
C00677=-119.480,-6.750,21.260,0.4300,0.0200,0.9000
C00678=-118.980,-12.920,21.270,0.4200,0.0400,0.9100
C00679=-118.430,-18.460,21.320,0.4100,0.0300,0.9100
C00680=-118.280,-22.180,21.460,0.3600,-0.0200,0.9300
C00681=-118.520,-24.730,21.640,0.2800,-0.0500,0.9600
C00682=-118.980,-26.820,21.810,0.1900,-0.0500,0.9800
C00683=-119.440,-28.930,21.940,0.1300,-0.0200,0.9900
C00684=-119.630,-31.560,22.000,0.0800,0.0000,1.0000
C00685=-119.350,-35.030,22.030,0.0300,0.0000,1.0000
C00686=-118.610,-38.910,22.060,0.0100,0.0000,1.0000
C00687=-117.470,-42.660,22.080,0.0000,0.0000,1.0000
C00688=-116.170,-46.140,22.100,0.0000,0.0000,1.0000
C00689=-114.770,-49.510,22.100,0.0000,0.0000,1.0000
C00690=-113.230,-52.890,22.080,0.0000,0.0000,1.0000
C00691=-111.380,-56.360,22.060,0.0100,0.0000,1.0000
C00692=-109.160,-59.620,22.030,0.0300,0.0200,1.0000
C00693=-106.900,-62.270,22.000,0.0500,0.0500,1.0000
C00694=-104.920,-64.000,21.940,0.0700,0.1000,0.9900
C00695=-103.090,-65.170,21.810,0.1000,0.1700,0.9800
C00696=-101.290,-66.320,21.640,0.1600,0.2300,0.9600
C00697=-99.320,-67.960,21.460,0.2400,0.2700,0.9300
C00698=-96.800,-70.690,21.320,0.3100,0.2700,0.9100
C00699=-93.270,-75.000,21.270,0.3300,0.2700,0.9100
C00700=-89.260,-79.710,21.260,0.3200,0.2800,0.9000
C00701=-84.620,-84.620,21.260,0.3000,0.3000,0.9000
C00702=-79.710,-89.260,21.260,0.2800,0.3200,0.9000
C00703=-75.000,-93.270,21.270,0.2700,0.3300,0.9100
C00704=-70.690,-96.800,21.320,0.2700,0.3100,0.9100
C00705=-67.960,-99.320,21.460,0.2700,0.2400,0.9300
C00706=-66.320,-101.290,21.640,0.2300,0.1600,0.9600
C00707=-65.170,-103.090,21.810,0.1700,0.1000,0.9800
C00708=-64.000,-104.920,21.940,0.1000,0.0700,0.9900
C00709=-62.270,-106.900,22.000,0.0500,0.0500,1.0000
C00710=-59.620,-109.160,22.030,0.0200,0.0300,1.0000
C00711=-56.360,-111.380,22.060,0.0000,0.0100,1.0000
C00712=-52.890,-113.230,22.080,0.0000,0.0000,1.0000
C00713=-49.510,-114.770,22.100,0.0000,0.0000,1.0000
C00714=-46.140,-116.170,22.100,0.0000,0.0000,1.0000
C00715=-42.660,-117.470,22.080,0.0000,0.0000,1.0000
C00716=-38.910,-118.610,22.060,0.0000,0.0100,1.0000
C00717=-35.030,-119.350,22.030,0.0000,0.0300,1.0000
C00718=-31.560,-119.630,22.000,0.0000,0.0800,1.0000
C00719=-28.930,-119.440,21.940,-0.0200,0.1300,0.9900
C00720=-26.820,-118.980,21.810,-0.0500,0.1900,0.9800
C00721=-24.730,-118.520,21.640,-0.0500,0.2800,0.9600
C00722=-22.180,-118.280,21.460,-0.0200,0.3600,0.9300
C00723=-18.460,-118.430,21.320,0.0300,0.4100,0.9100
C00724=-12.920,-118.980,21.270,0.0400,0.4200,0.9100
C00725=-6.750,-119.480,21.260,0.0200,0.4300,0.9000
C00726=0.000,-119.670,21.260,0.0000,0.4300,0.9000
C00727=0.000,-119.670,21.260,0.0000,0.4300,0.9000
C00728=6.750,-119.480,21.260,-0.0200,0.4300,0.9000
C00729=12.920,-118.980,21.270,-0.0400,0.4200,0.9100
C00730=18.460,-118.430,21.320,-0.0300,0.4100,0.9100
C00731=22.180,-118.280,21.460,0.0200,0.3600,0.9300
C00732=24.730,-118.520,21.640,0.0500,0.2800,0.9600
C00733=26.820,-118.980,21.810,0.0500,0.1900,0.9800
C00734=28.930,-119.440,21.940,0.0200,0.1300,0.9900
C00735=31.560,-119.630,22.000,-0.0000,0.0800,1.0000
C00736=35.030,-119.350,22.030,-0.0000,0.0300,1.0000
C00737=38.910,-118.610,22.060,-0.0000,0.0100,1.0000
C00738=42.660,-117.470,22.080,-0.0000,0.0000,1.0000
C00739=46.140,-116.170,22.100,-0.0000,0.0000,1.0000
C00740=49.510,-114.770,22.100,-0.0000,0.0000,1.0000
C00741=52.890,-113.230,22.080,-0.0000,0.0000,1.0000
C00742=56.360,-111.380,22.060,-0.0000,0.0100,1.0000
C00743=59.620,-109.160,22.030,-0.0200,0.0300,1.0000
C00744=62.270,-106.900,22.000,-0.0500,0.0500,1.0000
C00745=64.000,-104.920,21.940,-0.1000,0.0700,0.9900
C00746=65.170,-103.090,21.810,-0.1700,0.1000,0.9800
C00747=66.320,-101.290,21.640,-0.2300,0.1600,0.9600
C00748=67.960,-99.320,21.460,-0.2700,0.2400,0.9300
C00749=70.690,-96.800,21.320,-0.2700,0.3100,0.9100
C00750=75.000,-93.270,21.270,-0.2700,0.3300,0.9100
C00751=79.710,-89.260,21.260,-0.2800,0.3200,0.9000
C00752=84.620,-84.620,21.260,-0.3000,0.3000,0.9000
C00753=89.260,-79.710,21.260,-0.3200,0.2800,0.9000
C00754=93.270,-75.000,21.270,-0.3300,0.2700,0.9100
C00755=96.800,-70.690,21.320,-0.3100,0.2700,0.9100
C00756=99.320,-67.960,21.460,-0.2400,0.2700,0.9300
C00757=101.290,-66.320,21.640,-0.1600,0.2300,0.9600
C00758=103.090,-65.170,21.810,-0.1000,0.1700,0.9800
C00759=104.920,-64.000,21.940,-0.0700,0.1000,0.9900
C00760=106.900,-62.270,22.000,-0.0500,0.0500,1.0000
C00761=109.160,-59.620,22.030,-0.0300,0.0200,1.0000
C00762=111.380,-56.360,22.060,-0.0100,0.0000,1.0000
C00763=113.230,-52.890,22.080,-0.0000,0.0000,1.0000
C00764=114.770,-49.510,22.100,-0.0000,0.0000,1.0000
C00765=116.170,-46.140,22.100,-0.0000,0.0000,1.0000
C00766=117.470,-42.660,22.080,-0.0000,0.0000,1.0000
C00767=118.610,-38.910,22.060,-0.0100,0.0000,1.0000
C00768=119.350,-35.030,22.030,-0.0300,0.0000,1.0000
C00769=119.630,-31.560,22.000,-0.0800,0.0000,1.0000
C00770=119.440,-28.930,21.940,-0.1300,-0.0200,0.9900
C00771=118.980,-26.820,21.810,-0.1900,-0.0500,0.9800
C00772=118.520,-24.730,21.640,-0.2800,-0.0500,0.9600
C00773=118.280,-22.180,21.460,-0.3600,-0.0200,0.9300
C00774=118.430,-18.460,21.320,-0.4100,0.0300,0.9100
C00775=118.980,-12.920,21.270,-0.4200,0.0400,0.9100
C00776=119.480,-6.750,21.260,-0.4300,0.0200,0.9000
C00777=119.670,0.000,21.260,-0.4300,0.0000,0.9000
C00778=119.480,6.750,21.260,-0.4300,-0.0200,0.9000
C00779=118.980,12.920,21.270,-0.4200,-0.0400,0.9100
C00780=118.430,18.460,21.320,-0.4100,-0.0300,0.9100
C00781=118.280,22.180,21.460,-0.3600,0.0200,0.9300
C00782=118.520,24.730,21.640,-0.2800,0.0500,0.9600
C00783=118.980,26.820,21.810,-0.1900,0.0500,0.9800
C00784=119.440,28.930,21.940,-0.1300,0.0200,0.9900
C00785=119.630,31.560,22.000,-0.0800,-0.0000,1.0000
C00786=119.350,35.030,22.030,-0.0300,-0.0000,1.0000
C00787=118.610,38.910,22.060,-0.0100,-0.0000,1.0000
C00788=117.470,42.660,22.080,-0.0000,-0.0000,1.0000
C00789=116.170,46.140,22.100,-0.0000,-0.0000,1.0000
C00790=114.770,49.510,22.100,-0.0000,-0.0000,1.0000
C00791=113.230,52.890,22.080,-0.0000,-0.0000,1.0000
C00792=111.380,56.360,22.060,-0.0100,-0.0000,1.0000
C00793=109.160,59.620,22.030,-0.0300,-0.0200,1.0000
C00794=106.900,62.270,22.000,-0.0500,-0.0500,1.0000
C00795=104.920,64.000,21.940,-0.0700,-0.1000,0.9900
C00796=103.090,65.170,21.810,-0.1000,-0.1700,0.9800
C00797=101.290,66.320,21.640,-0.1600,-0.2300,0.9600
C00798=99.320,67.960,21.460,-0.2400,-0.2700,0.9300
C00799=96.800,70.690,21.320,-0.3100,-0.2700,0.9100
C00800=93.270,75.000,21.270,-0.3300,-0.2700,0.9100
C00801=89.260,79.710,21.260,-0.3200,-0.2800,0.9000
C00802=84.620,84.620,21.260,-0.3000,-0.3000,0.9000
C00803=79.710,89.260,21.260,-0.2800,-0.3200,0.9000
C00804=75.000,93.270,21.270,-0.2700,-0.3300,0.9100
C00805=70.690,96.800,21.320,-0.2700,-0.3100,0.9100
C00806=67.960,99.320,21.460,-0.2700,-0.2400,0.9300
C00807=66.320,101.290,21.640,-0.2300,-0.1600,0.9600
C00808=65.170,103.090,21.810,-0.1700,-0.1000,0.9800
C00809=64.000,104.920,21.940,-0.1000,-0.0700,0.9900
C00810=62.270,106.900,22.000,-0.0500,-0.0500,1.0000
C00811=59.620,109.160,22.030,-0.0200,-0.0300,1.0000
C00812=56.360,111.380,22.060,-0.0000,-0.0100,1.0000
C00813=52.890,113.230,22.080,-0.0000,-0.0000,1.0000
C00814=49.510,114.770,22.100,-0.0000,-0.0000,1.0000
C00815=46.140,116.170,22.100,-0.0000,-0.0000,1.0000
C00816=42.660,117.470,22.080,-0.0000,-0.0000,1.0000
C00817=38.910,118.610,22.060,-0.0000,-0.0100,1.0000
C00818=35.030,119.350,22.030,-0.0000,-0.0300,1.0000
C00819=31.560,119.630,22.000,-0.0000,-0.0800,1.0000
C00820=28.930,119.440,21.940,0.0200,-0.1300,0.9900
C00821=26.820,118.980,21.810,0.0500,-0.1900,0.9800
C00822=24.730,118.520,21.640,0.0500,-0.2800,0.9600
C00823=22.180,118.280,21.460,0.0200,-0.3600,0.9300
C00824=18.460,118.430,21.320,-0.0300,-0.4100,0.9100
C00825=12.920,118.980,21.270,-0.0400,-0.4200,0.9100
C00826=6.750,119.480,21.260,-0.0200,-0.4300,0.9000
C00827=0.000,119.670,21.260,0.0000,-0.4300,0.9000
C00828=0.000,118.930,22.800,0.0000,-0.4400,0.9000
C00829=6.690,118.740,22.790,-0.0300,-0.4400,0.9000
C00830=12.800,118.250,22.800,-0.0400,-0.4400,0.9000
C00831=18.320,117.730,22.860,-0.0300,-0.4300,0.9000
C00832=22.010,117.650,23.030,0.0300,-0.3700,0.9300
C00833=24.540,117.990,23.240,0.0700,-0.2800,0.9600
C00834=26.610,118.580,23.450,0.0600,-0.1800,0.9800
C00835=28.710,119.180,23.600,0.0300,-0.1200,0.9900
C00836=31.320,119.500,23.680,0.0000,-0.0700,1.0000
C00837=34.810,119.320,23.720,-0.0000,-0.0300,1.0000
C00838=38.730,118.640,23.750,-0.0000,-0.0100,1.0000
C00839=42.550,117.500,23.780,-0.0000,-0.0000,1.0000
C00840=46.110,116.180,23.800,-0.0000,-0.0000,1.0000
C00841=49.550,114.760,23.800,-0.0000,-0.0000,1.0000
C00842=53.000,113.170,23.780,-0.0000,-0.0000,1.0000
C00843=56.500,111.280,23.750,-0.0000,-0.0000,1.0000
C00844=59.760,108.990,23.720,-0.0200,-0.0200,1.0000
C00845=62.350,106.640,23.680,-0.0500,-0.0500,1.0000
C00846=63.970,104.580,23.600,-0.1100,-0.0700,0.9900
C00847=65.030,102.660,23.450,-0.1700,-0.0900,0.9800
C00848=66.080,100.780,23.240,-0.2500,-0.1500,0.9600
C00849=67.630,98.750,23.030,-0.2900,-0.2400,0.9300
C00850=70.290,96.200,22.860,-0.2800,-0.3200,0.9000
C00851=74.560,92.670,22.800,-0.2800,-0.3400,0.9000
C00852=79.240,88.690,22.790,-0.3000,-0.3300,0.9000
C00853=84.100,84.100,22.800,-0.3100,-0.3100,0.9000
C00854=88.690,79.240,22.790,-0.3300,-0.3000,0.9000
C00855=92.670,74.560,22.800,-0.3400,-0.2800,0.9000
C00856=96.200,70.290,22.860,-0.3200,-0.2800,0.9000
C00857=98.750,67.630,23.030,-0.2400,-0.2900,0.9300
C00858=100.780,66.080,23.240,-0.1500,-0.2500,0.9600
C00859=102.660,65.030,23.450,-0.0900,-0.1700,0.9800
C00860=104.580,63.970,23.600,-0.0700,-0.1100,0.9900
C00861=106.640,62.350,23.680,-0.0500,-0.0500,1.0000
C00862=108.990,59.760,23.720,-0.0200,-0.0200,1.0000
C00863=111.280,56.500,23.750,-0.0000,-0.0000,1.0000
C00864=113.170,53.000,23.780,-0.0000,-0.0000,1.0000
C00865=114.760,49.550,23.800,-0.0000,-0.0000,1.0000
C00866=116.180,46.110,23.800,-0.0000,-0.0000,1.0000
C00867=117.500,42.550,23.780,-0.0000,-0.0000,1.0000
C00868=118.640,38.730,23.750,-0.0100,-0.0000,1.0000
C00869=119.320,34.810,23.720,-0.0300,-0.0000,1.0000
C00870=119.500,31.320,23.680,-0.0700,0.0000,1.0000
C00871=119.180,28.710,23.600,-0.1200,0.0300,0.9900
C00872=118.580,26.610,23.450,-0.1800,0.0600,0.9800
C00873=117.990,24.540,23.240,-0.2800,0.0700,0.9600
C00874=117.650,22.010,23.030,-0.3700,0.0300,0.9300
C00875=117.730,18.320,22.860,-0.4300,-0.0300,0.9000
C00876=118.250,12.800,22.800,-0.4400,-0.0400,0.9000
C00877=118.740,6.690,22.790,-0.4400,-0.0300,0.9000
C00878=118.930,0.000,22.800,-0.4400,0.0000,0.9000
C00879=118.740,-6.690,22.790,-0.4400,0.0300,0.9000
C00880=118.250,-12.800,22.800,-0.4400,0.0400,0.9000
C00881=117.730,-18.320,22.860,-0.4300,0.0300,0.9000
C00882=117.650,-22.010,23.030,-0.3700,-0.0300,0.9300
C00883=117.990,-24.540,23.240,-0.2800,-0.0700,0.9600
C00884=118.580,-26.610,23.450,-0.1800,-0.0600,0.9800
C00885=119.180,-28.710,23.600,-0.1200,-0.0300,0.9900
C00886=119.500,-31.320,23.680,-0.0700,-0.0000,1.0000
C00887=119.320,-34.810,23.720,-0.0300,0.0000,1.0000
C00888=118.640,-38.730,23.750,-0.0100,0.0000,1.0000
C00889=117.500,-42.550,23.780,-0.0000,0.0000,1.0000
C00890=116.180,-46.110,23.800,-0.0000,0.0000,1.0000
C00891=114.760,-49.550,23.800,-0.0000,0.0000,1.0000
C00892=113.170,-53.000,23.780,-0.0000,0.0000,1.0000
C00893=111.280,-56.500,23.750,-0.0000,0.0000,1.0000
C00894=108.990,-59.760,23.720,-0.0200,0.0200,1.0000
C00895=106.640,-62.350,23.680,-0.0500,0.0500,1.0000
C00896=104.580,-63.970,23.600,-0.0700,0.1100,0.9900
C00897=102.660,-65.030,23.450,-0.0900,0.1700,0.9800
C00898=100.780,-66.080,23.240,-0.1500,0.2500,0.9600
C00899=98.750,-67.630,23.030,-0.2400,0.2900,0.9300
C00900=96.200,-70.290,22.860,-0.3200,0.2800,0.9000
C00901=92.670,-74.560,22.800,-0.3400,0.2800,0.9000
C00902=88.690,-79.240,22.790,-0.3300,0.3000,0.9000
C00903=84.100,-84.100,22.800,-0.3100,0.3100,0.9000
C00904=79.240,-88.690,22.790,-0.3000,0.3300,0.9000
C00905=74.560,-92.670,22.800,-0.2800,0.3400,0.9000
C00906=70.290,-96.200,22.860,-0.2800,0.3200,0.9000
C00907=67.630,-98.750,23.030,-0.2900,0.2400,0.9300
C00908=66.080,-100.780,23.240,-0.2500,0.1500,0.9600
C00909=65.030,-102.660,23.450,-0.1700,0.0900,0.9800
C00910=63.970,-104.580,23.600,-0.1100,0.0700,0.9900
C00911=62.350,-106.640,23.680,-0.0500,0.0500,1.0000
C00912=59.760,-108.990,23.720,-0.0200,0.0200,1.0000
C00913=56.500,-111.280,23.750,-0.0000,0.0000,1.0000
C00914=53.000,-113.170,23.780,-0.0000,0.0000,1.0000
C00915=49.550,-114.760,23.800,-0.0000,0.0000,1.0000
C00916=46.110,-116.180,23.800,-0.0000,0.0000,1.0000
C00917=42.550,-117.500,23.780,-0.0000,0.0000,1.0000
C00918=38.730,-118.640,23.750,-0.0000,0.0100,1.0000
C00919=34.810,-119.320,23.720,-0.0000,0.0300,1.0000
C00920=31.320,-119.500,23.680,0.0000,0.0700,1.0000
C00921=28.710,-119.180,23.600,0.0300,0.1200,0.9900
C00922=26.610,-118.580,23.450,0.0600,0.1800,0.9800
C00923=24.540,-117.990,23.240,0.0700,0.2800,0.9600
C00924=22.010,-117.650,23.030,0.0300,0.3700,0.9300
C00925=18.320,-117.730,22.860,-0.0300,0.4300,0.9000
C00926=12.800,-118.250,22.800,-0.0400,0.4400,0.9000
C00927=6.690,-118.740,22.790,-0.0300,0.4400,0.9000
C00928=0.000,-118.930,22.800,0.0000,0.4400,0.9000
C00929=0.000,-118.930,22.800,0.0000,0.4400,0.9000
C00930=-6.690,-118.740,22.790,0.0300,0.4400,0.9000
C00931=-12.800,-118.250,22.800,0.0400,0.4400,0.9000
C00932=-18.320,-117.730,22.860,0.0300,0.4300,0.9000
C00933=-22.010,-117.650,23.030,-0.0300,0.3700,0.9300
C00934=-24.540,-117.990,23.240,-0.0700,0.2800,0.9600
C00935=-26.610,-118.580,23.450,-0.0600,0.1800,0.9800
C00936=-28.710,-119.180,23.600,-0.0300,0.1200,0.9900
C00937=-31.320,-119.500,23.680,-0.0000,0.0700,1.0000
C00938=-34.810,-119.320,23.720,0.0000,0.0300,1.0000
C00939=-38.730,-118.640,23.750,0.0000,0.0100,1.0000
C00940=-42.550,-117.500,23.780,0.0000,0.0000,1.0000
C00941=-46.110,-116.180,23.800,0.0000,0.0000,1.0000
C00942=-49.550,-114.760,23.800,0.0000,0.0000,1.0000
C00943=-53.000,-113.170,23.780,0.0000,0.0000,1.0000
C00944=-56.500,-111.280,23.750,0.0000,0.0000,1.0000
C00945=-59.760,-108.990,23.720,0.0200,0.0200,1.0000
C00946=-62.350,-106.640,23.680,0.0500,0.0500,1.0000
C00947=-63.970,-104.580,23.600,0.1100,0.0700,0.9900
C00948=-65.030,-102.660,23.450,0.1700,0.0900,0.9800
C00949=-66.080,-100.780,23.240,0.2500,0.1500,0.9600
C00950=-67.630,-98.750,23.030,0.2900,0.2400,0.9300
C00951=-70.290,-96.200,22.860,0.2800,0.3200,0.9000
C00952=-74.560,-92.670,22.800,0.2800,0.3400,0.9000
C00953=-79.240,-88.690,22.790,0.3000,0.3300,0.9000
C00954=-84.100,-84.100,22.800,0.3100,0.3100,0.9000
C00955=-88.690,-79.240,22.790,0.3300,0.3000,0.9000
C00956=-92.670,-74.560,22.800,0.3400,0.2800,0.9000
C00957=-96.200,-70.290,22.860,0.3200,0.2800,0.9000
C00958=-98.750,-67.630,23.030,0.2400,0.2900,0.9300
C00959=-100.780,-66.080,23.240,0.1500,0.2500,0.9600
C00960=-102.660,-65.030,23.450,0.0900,0.1700,0.9800
C00961=-104.580,-63.970,23.600,0.0700,0.1100,0.9900
C00962=-106.640,-62.350,23.680,0.0500,0.0500,1.0000
C00963=-108.990,-59.760,23.720,0.0200,0.0200,1.0000
C00964=-111.280,-56.500,23.750,0.0000,0.0000,1.0000
C00965=-113.170,-53.000,23.780,0.0000,0.0000,1.0000
C00966=-114.760,-49.550,23.800,0.0000,0.0000,1.0000
C00967=-116.180,-46.110,23.800,0.0000,0.0000,1.0000
C00968=-117.500,-42.550,23.780,0.0000,0.0000,1.0000
C00969=-118.640,-38.730,23.750,0.0100,0.0000,1.0000
C00970=-119.320,-34.810,23.720,0.0300,0.0000,1.0000
C00971=-119.500,-31.320,23.680,0.0700,-0.0000,1.0000
C00972=-119.180,-28.710,23.600,0.1200,-0.0300,0.9900
C00973=-118.580,-26.610,23.450,0.1800,-0.0600,0.9800
C00974=-117.990,-24.540,23.240,0.2800,-0.0700,0.9600
C00975=-117.650,-22.010,23.030,0.3700,-0.0300,0.9300
C00976=-117.730,-18.320,22.860,0.4300,0.0300,0.9000
C00977=-118.250,-12.800,22.800,0.4400,0.0400,0.9000
C00978=-118.740,-6.690,22.790,0.4400,0.0300,0.9000
C00979=-118.930,0.000,22.800,0.4400,-0.0000,0.9000
C00980=-118.740,6.690,22.790,0.4400,-0.0300,0.9000
C00981=-118.250,12.800,22.800,0.4400,-0.0400,0.9000
C00982=-117.730,18.320,22.860,0.4300,-0.0300,0.9000
C00983=-117.650,22.010,23.030,0.3700,0.0300,0.9300
C00984=-117.990,24.540,23.240,0.2800,0.0700,0.9600
C00985=-118.580,26.610,23.450,0.1800,0.0600,0.9800
C00986=-119.180,28.710,23.600,0.1200,0.0300,0.9900
C00987=-119.500,31.320,23.680,0.0700,0.0000,1.0000
C00988=-119.320,34.810,23.720,0.0300,-0.0000,1.0000
C00989=-118.640,38.730,23.750,0.0100,-0.0000,1.0000
C00990=-117.500,42.550,23.780,0.0000,-0.0000,1.0000
C00991=-116.180,46.110,23.800,0.0000,-0.0000,1.0000
C00992=-114.760,49.550,23.800,0.0000,-0.0000,1.0000
C00993=-113.170,53.000,23.780,0.0000,-0.0000,1.0000
C00994=-111.280,56.500,23.750,0.0000,-0.0000,1.0000
C00995=-108.990,59.760,23.720,0.0200,-0.0200,1.0000
C00996=-106.640,62.350,23.680,0.0500,-0.0500,1.0000
C00997=-104.580,63.970,23.600,0.0700,-0.1100,0.9900
C00998=-102.660,65.030,23.450,0.0900,-0.1700,0.9800
C00999=-100.780,66.080,23.240,0.1500,-0.2500,0.9600
C01000=-98.750,67.630,23.030,0.2400,-0.2900,0.9300
C01001=-96.200,70.290,22.860,0.3200,-0.2800,0.9000
C01002=-92.670,74.560,22.800,0.3400,-0.2800,0.9000
C01003=-88.690,79.240,22.790,0.3300,-0.3000,0.9000
C01004=-84.100,84.100,22.800,0.3100,-0.3100,0.9000
C01005=-79.240,88.690,22.790,0.3000,-0.3300,0.9000
C01006=-74.560,92.670,22.800,0.2800,-0.3400,0.9000
C01007=-70.290,96.200,22.860,0.2800,-0.3200,0.9000
C01008=-67.630,98.750,23.030,0.2900,-0.2400,0.9300
C01009=-66.080,100.780,23.240,0.2500,-0.1500,0.9600
C01010=-65.030,102.660,23.450,0.1700,-0.0900,0.9800
C01011=-63.970,104.580,23.600,0.1100,-0.0700,0.9900
C01012=-62.350,106.640,23.680,0.0500,-0.0500,1.0000
C01013=-59.760,108.990,23.720,0.0200,-0.0200,1.0000
C01014=-56.500,111.280,23.750,0.0000,-0.0000,1.0000
C01015=-53.000,113.170,23.780,0.0000,-0.0000,1.0000
C01016=-49.550,114.760,23.800,0.0000,-0.0000,1.0000
C01017=-46.110,116.180,23.800,0.0000,-0.0000,1.0000
C01018=-42.550,117.500,23.780,0.0000,-0.0000,1.0000
C01019=-38.730,118.640,23.750,0.0000,-0.0100,1.0000
C01020=-34.810,119.320,23.720,0.0000,-0.0300,1.0000
C01021=-31.320,119.500,23.680,-0.0000,-0.0700,1.0000
C01022=-28.710,119.180,23.600,-0.0300,-0.1200,0.9900
C01023=-26.610,118.580,23.450,-0.0600,-0.1800,0.9800
C01024=-24.540,117.990,23.240,-0.0700,-0.2800,0.9600
C01025=-22.010,117.650,23.030,-0.0300,-0.3700,0.9300
C01026=-18.320,117.730,22.860,0.0300,-0.4300,0.9000
C01027=-12.800,118.250,22.800,0.0400,-0.4400,0.9000
C01028=-6.690,118.740,22.790,0.0300,-0.4400,0.9000
C01029=0.000,118.930,22.800,0.0000,-0.4400,0.9000
C01030=0.000,118.160,24.310,0.0000,-0.4600,0.8900
C01031=-6.620,117.970,24.310,0.0300,-0.4600,0.8900
C01032=-12.680,117.490,24.310,0.0400,-0.4600,0.8900
C01033=-18.180,116.990,24.390,0.0200,-0.4400,0.9000
C01034=-21.830,116.980,24.580,-0.0500,-0.3800,0.9200
C01035=-24.340,117.430,24.840,-0.0900,-0.2800,0.9600
C01036=-26.390,118.160,25.080,-0.0700,-0.1700,0.9800
C01037=-28.480,118.910,25.270,-0.0300,-0.1200,0.9900
C01038=-31.070,119.360,25.350,-0.0100,-0.0700,1.0000
C01039=-34.570,119.290,25.400,0.0000,-0.0300,1.0000
C01040=-38.540,118.670,25.440,0.0000,-0.0000,1.0000
C01041=-42.430,117.540,25.470,0.0000,-0.0000,1.0000
C01042=-46.070,116.200,25.500,0.0000,-0.0000,1.0000
C01043=-49.590,114.740,25.500,0.0000,-0.0000,1.0000
C01044=-53.110,113.120,25.470,0.0000,-0.0000,1.0000
C01045=-56.660,111.170,25.440,0.0000,-0.0000,1.0000
C01046=-59.910,108.800,25.400,0.0200,-0.0200,1.0000
C01047=-62.430,106.370,25.350,0.0500,-0.0500,1.0000
C01048=-63.940,104.220,25.270,0.1100,-0.0600,0.9900
C01049=-64.890,102.210,25.080,0.1700,-0.0700,0.9800
C01050=-65.830,100.250,24.840,0.2600,-0.1300,0.9600
C01051=-67.280,98.160,24.580,0.3100,-0.2400,0.9200
C01052=-69.870,95.580,24.390,0.3000,-0.3300,0.9000
C01053=-74.110,92.050,24.310,0.2900,-0.3600,0.8900
C01054=-78.740,88.100,24.310,0.3100,-0.3500,0.8900
C01055=-83.550,83.550,24.310,0.3300,-0.3300,0.8900
C01056=-88.100,78.740,24.310,0.3500,-0.3100,0.8900
C01057=-92.050,74.110,24.310,0.3600,-0.2900,0.8900
C01058=-95.580,69.870,24.390,0.3300,-0.3000,0.9000
C01059=-98.160,67.280,24.580,0.2400,-0.3100,0.9200
C01060=-100.250,65.830,24.840,0.1300,-0.2600,0.9600
C01061=-102.210,64.890,25.080,0.0700,-0.1700,0.9800
C01062=-104.220,63.940,25.270,0.0600,-0.1100,0.9900
C01063=-106.370,62.430,25.350,0.0500,-0.0500,1.0000
C01064=-108.800,59.910,25.400,0.0200,-0.0200,1.0000
C01065=-111.170,56.660,25.440,0.0000,-0.0000,1.0000
C01066=-113.120,53.110,25.470,0.0000,-0.0000,1.0000
C01067=-114.740,49.590,25.500,0.0000,-0.0000,1.0000
C01068=-116.200,46.070,25.500,0.0000,-0.0000,1.0000
C01069=-117.540,42.430,25.470,0.0000,-0.0000,1.0000
C01070=-118.670,38.540,25.440,0.0000,-0.0000,1.0000
C01071=-119.290,34.570,25.400,0.0300,-0.0000,1.0000
C01072=-119.360,31.070,25.350,0.0700,0.0100,1.0000
C01073=-118.910,28.480,25.270,0.1200,0.0300,0.9900
C01074=-118.160,26.390,25.080,0.1700,0.0700,0.9800
C01075=-117.430,24.340,24.840,0.2800,0.0900,0.9600
C01076=-116.980,21.830,24.580,0.3800,0.0500,0.9200
C01077=-116.990,18.180,24.390,0.4400,-0.0200,0.9000
C01078=-117.490,12.680,24.310,0.4600,-0.0400,0.8900
C01079=-117.970,6.620,24.310,0.4600,-0.0300,0.8900
C01080=-118.160,0.000,24.310,0.4600,-0.0000,0.8900
C01081=-117.970,-6.620,24.310,0.4600,0.0300,0.8900
C01082=-117.490,-12.680,24.310,0.4600,0.0400,0.8900
C01083=-116.990,-18.180,24.390,0.4400,0.0200,0.9000
C01084=-116.980,-21.830,24.580,0.3800,-0.0500,0.9200
C01085=-117.430,-24.340,24.840,0.2800,-0.0900,0.9600
C01086=-118.160,-26.390,25.080,0.1700,-0.0700,0.9800
C01087=-118.910,-28.480,25.270,0.1200,-0.0300,0.9900
C01088=-119.360,-31.070,25.350,0.0700,-0.0100,1.0000
C01089=-119.290,-34.570,25.400,0.0300,0.0000,1.0000
C01090=-118.670,-38.540,25.440,0.0000,0.0000,1.0000
C01091=-117.540,-42.430,25.470,0.0000,0.0000,1.0000
C01092=-116.200,-46.070,25.500,0.0000,0.0000,1.0000
C01093=-114.740,-49.590,25.500,0.0000,0.0000,1.0000
C01094=-113.120,-53.110,25.470,0.0000,0.0000,1.0000
C01095=-111.170,-56.660,25.440,0.0000,0.0000,1.0000
C01096=-108.800,-59.910,25.400,0.0200,0.0200,1.0000
C01097=-106.370,-62.430,25.350,0.0500,0.0500,1.0000
C01098=-104.220,-63.940,25.270,0.0600,0.1100,0.9900
C01099=-102.210,-64.890,25.080,0.0700,0.1700,0.9800
C01100=-100.250,-65.830,24.840,0.1300,0.2600,0.9600
C01101=-98.160,-67.280,24.580,0.2400,0.3100,0.9200
C01102=-95.580,-69.870,24.390,0.3300,0.3000,0.9000
C01103=-92.050,-74.110,24.310,0.3600,0.2900,0.8900
C01104=-88.100,-78.740,24.310,0.3500,0.3100,0.8900
C01105=-83.550,-83.550,24.310,0.3300,0.3300,0.8900
C01106=-78.740,-88.100,24.310,0.3100,0.3500,0.8900
C01107=-74.110,-92.050,24.310,0.2900,0.3600,0.8900
C01108=-69.870,-95.580,24.390,0.3000,0.3300,0.9000
C01109=-67.280,-98.160,24.580,0.3100,0.2400,0.9200
C01110=-65.830,-100.250,24.840,0.2600,0.1300,0.9600
C01111=-64.890,-102.210,25.080,0.1700,0.0700,0.9800
C01112=-63.940,-104.220,25.270,0.1100,0.0600,0.9900
C01113=-62.430,-106.370,25.350,0.0500,0.0500,1.0000
C01114=-59.910,-108.800,25.400,0.0200,0.0200,1.0000
C01115=-56.660,-111.170,25.440,0.0000,0.0000,1.0000
C01116=-53.110,-113.120,25.470,0.0000,0.0000,1.0000
C01117=-49.590,-114.740,25.500,0.0000,0.0000,1.0000
C01118=-46.070,-116.200,25.500,0.0000,0.0000,1.0000
C01119=-42.430,-117.540,25.470,0.0000,0.0000,1.0000
C01120=-38.540,-118.670,25.440,0.0000,0.0000,1.0000
C01121=-34.570,-119.290,25.400,0.0000,0.0300,1.0000
C01122=-31.070,-119.360,25.350,-0.0100,0.0700,1.0000
C01123=-28.480,-118.910,25.270,-0.0300,0.1200,0.9900
C01124=-26.390,-118.160,25.080,-0.0700,0.1700,0.9800
C01125=-24.340,-117.430,24.840,-0.0900,0.2800,0.9600
C01126=-21.830,-116.980,24.580,-0.0500,0.3800,0.9200
C01127=-18.180,-116.990,24.390,0.0200,0.4400,0.9000
C01128=-12.680,-117.490,24.310,0.0400,0.4600,0.8900
C01129=-6.620,-117.970,24.310,0.0300,0.4600,0.8900
C01130=0.000,-118.160,24.310,0.0000,0.4600,0.8900
C01131=0.000,-118.160,24.310,0.0000,0.4600,0.8900
C01132=6.620,-117.970,24.310,-0.0300,0.4600,0.8900
C01133=12.680,-117.490,24.310,-0.0400,0.4600,0.8900
C01134=18.180,-116.990,24.390,-0.0200,0.4400,0.9000
C01135=21.830,-116.980,24.580,0.0500,0.3800,0.9200
C01136=24.340,-117.430,24.840,0.0900,0.2800,0.9600
C01137=26.390,-118.160,25.080,0.0700,0.1700,0.9800
C01138=28.480,-118.910,25.270,0.0300,0.1200,0.9900
C01139=31.070,-119.360,25.350,0.0100,0.0700,1.0000
C01140=34.570,-119.290,25.400,-0.0000,0.0300,1.0000
C01141=38.540,-118.670,25.440,-0.0000,0.0000,1.0000
C01142=42.430,-117.540,25.470,-0.0000,0.0000,1.0000
C01143=46.070,-116.200,25.500,-0.0000,0.0000,1.0000
C01144=49.590,-114.740,25.500,-0.0000,0.0000,1.0000
C01145=53.110,-113.120,25.470,-0.0000,0.0000,1.0000
C01146=56.660,-111.170,25.440,-0.0000,0.0000,1.0000
C01147=59.910,-108.800,25.400,-0.0200,0.0200,1.0000
C01148=62.430,-106.370,25.350,-0.0500,0.0500,1.0000
C01149=63.940,-104.220,25.270,-0.1100,0.0600,0.9900
C01150=64.890,-102.210,25.080,-0.1700,0.0700,0.9800
C01151=65.830,-100.250,24.840,-0.2600,0.1300,0.9600
C01152=67.280,-98.160,24.580,-0.3100,0.2400,0.9200
C01153=69.870,-95.580,24.390,-0.3000,0.3300,0.9000
C01154=74.110,-92.050,24.310,-0.2900,0.3600,0.8900
C01155=78.740,-88.100,24.310,-0.3100,0.3500,0.8900
C01156=83.550,-83.550,24.310,-0.3300,0.3300,0.8900
C01157=88.100,-78.740,24.310,-0.3500,0.3100,0.8900
C01158=92.050,-74.110,24.310,-0.3600,0.2900,0.8900
C01159=95.580,-69.870,24.390,-0.3300,0.3000,0.9000
C01160=98.160,-67.280,24.580,-0.2400,0.3100,0.9200
C01161=100.250,-65.830,24.840,-0.1300,0.2600,0.9600
C01162=102.210,-64.890,25.080,-0.0700,0.1700,0.9800
C01163=104.220,-63.940,25.270,-0.0600,0.1100,0.9900
C01164=106.370,-62.430,25.350,-0.0500,0.0500,1.0000
C01165=108.800,-59.910,25.400,-0.0200,0.0200,1.0000
C01166=111.170,-56.660,25.440,-0.0000,0.0000,1.0000
C01167=113.120,-53.110,25.470,-0.0000,0.0000,1.0000
C01168=114.740,-49.590,25.500,-0.0000,0.0000,1.0000
C01169=116.200,-46.070,25.500,-0.0000,0.0000,1.0000
C01170=117.540,-42.430,25.470,-0.0000,0.0000,1.0000
C01171=118.670,-38.540,25.440,-0.0000,0.0000,1.0000
C01172=119.290,-34.570,25.400,-0.0300,0.0000,1.0000
C01173=119.360,-31.070,25.350,-0.0700,-0.0100,1.0000
C01174=118.910,-28.480,25.270,-0.1200,-0.0300,0.9900
C01175=118.160,-26.390,25.080,-0.1700,-0.0700,0.9800
C01176=117.430,-24.340,24.840,-0.2800,-0.0900,0.9600
C01177=116.980,-21.830,24.580,-0.3800,-0.0500,0.9200
C01178=116.990,-18.180,24.390,-0.4400,0.0200,0.9000
C01179=117.490,-12.680,24.310,-0.4600,0.0400,0.8900
C01180=117.970,-6.620,24.310,-0.4600,0.0300,0.8900
C01181=118.160,0.000,24.310,-0.4600,0.0000,0.8900
C01182=117.970,6.620,24.310,-0.4600,-0.0300,0.8900
C01183=117.490,12.680,24.310,-0.4600,-0.0400,0.8900
C01184=116.990,18.180,24.390,-0.4400,-0.0200,0.9000
C01185=116.980,21.830,24.580,-0.3800,0.0500,0.9200
C01186=117.430,24.340,24.840,-0.2800,0.0900,0.9600
C01187=118.160,26.390,25.080,-0.1700,0.0700,0.9800
C01188=118.910,28.480,25.270,-0.1200,0.0300,0.9900
C01189=119.360,31.070,25.350,-0.0700,0.0100,1.0000
C01190=119.290,34.570,25.400,-0.0300,-0.0000,1.0000
C01191=118.670,38.540,25.440,-0.0000,-0.0000,1.0000
C01192=117.540,42.430,25.470,-0.0000,-0.0000,1.0000
C01193=116.200,46.070,25.500,-0.0000,-0.0000,1.0000
C01194=114.740,49.590,25.500,-0.0000,-0.0000,1.0000
C01195=113.120,53.110,25.470,-0.0000,-0.0000,1.0000
C01196=111.170,56.660,25.440,-0.0000,-0.0000,1.0000
C01197=108.800,59.910,25.400,-0.0200,-0.0200,1.0000
C01198=106.370,62.430,25.350,-0.0500,-0.0500,1.0000
C01199=104.220,63.940,25.270,-0.0600,-0.1100,0.9900
C01200=102.210,64.890,25.080,-0.0700,-0.1700,0.9800
C01201=100.250,65.830,24.840,-0.1300,-0.2600,0.9600
C01202=98.160,67.280,24.580,-0.2400,-0.3100,0.9200
C01203=95.580,69.870,24.390,-0.3300,-0.3000,0.9000
C01204=92.050,74.110,24.310,-0.3600,-0.2900,0.8900
C01205=88.100,78.740,24.310,-0.3500,-0.3100,0.8900
C01206=83.550,83.550,24.310,-0.3300,-0.3300,0.8900
C01207=78.740,88.100,24.310,-0.3100,-0.3500,0.8900
C01208=74.110,92.050,24.310,-0.2900,-0.3600,0.8900
C01209=69.870,95.580,24.390,-0.3000,-0.3300,0.9000
C01210=67.280,98.160,24.580,-0.3100,-0.2400,0.9200
C01211=65.830,100.250,24.840,-0.2600,-0.1300,0.9600
C01212=64.890,102.210,25.080,-0.1700,-0.0700,0.9800
C01213=63.940,104.220,25.270,-0.1100,-0.0600,0.9900
C01214=62.430,106.370,25.350,-0.0500,-0.0500,1.0000
C01215=59.910,108.800,25.400,-0.0200,-0.0200,1.0000
C01216=56.660,111.170,25.440,-0.0000,-0.0000,1.0000
C01217=53.110,113.120,25.470,-0.0000,-0.0000,1.0000
C01218=49.590,114.740,25.500,-0.0000,-0.0000,1.0000
C01219=46.070,116.200,25.500,-0.0000,-0.0000,1.0000
C01220=42.430,117.540,25.470,-0.0000,-0.0000,1.0000
C01221=38.540,118.670,25.440,-0.0000,-0.0000,1.0000
C01222=34.570,119.290,25.400,-0.0000,-0.0300,1.0000
C01223=31.070,119.360,25.350,0.0100,-0.0700,1.0000
C01224=28.480,118.910,25.270,0.0300,-0.1200,0.9900
C01225=26.390,118.160,25.080,0.0700,-0.1700,0.9800
C01226=24.340,117.430,24.840,0.0900,-0.2800,0.9600
C01227=21.830,116.980,24.580,0.0500,-0.3800,0.9200
C01228=18.180,116.990,24.390,-0.0200,-0.4400,0.9000
C01229=12.680,117.490,24.310,-0.0400,-0.4600,0.8900
C01230=6.620,117.970,24.310,-0.0300,-0.4600,0.8900
C01231=0.000,118.160,24.310,0.0000,-0.4600,0.8900
C01232=0.000,117.360,25.810,0.0000,-0.4800,0.8800
C01233=6.540,117.170,25.810,-0.0300,-0.4800,0.8800
C01234=12.560,116.700,25.810,-0.0400,-0.4800,0.8800
C01235=18.030,116.230,25.900,-0.0200,-0.4600,0.8900
C01236=21.650,116.290,26.130,0.0600,-0.3900,0.9200
C01237=24.130,116.850,26.420,0.1000,-0.2700,0.9600
C01238=26.170,117.720,26.710,0.0800,-0.1600,0.9800
C01239=28.240,118.620,26.920,0.0400,-0.1100,0.9900
C01240=30.810,119.220,27.030,0.0100,-0.0700,1.0000
C01241=34.320,119.260,27.080,-0.0000,-0.0300,1.0000
C01242=38.350,118.710,27.120,-0.0000,-0.0000,1.0000
C01243=42.310,117.580,27.170,-0.0000,-0.0000,1.0000
C01244=46.020,116.210,27.200,-0.0000,-0.0000,1.0000
C01245=49.630,114.720,27.200,-0.0000,-0.0000,1.0000
C01246=53.230,113.060,27.170,-0.0000,-0.0000,1.0000
C01247=56.820,111.060,27.120,-0.0000,-0.0000,1.0000
C01248=60.060,108.600,27.080,-0.0200,-0.0200,1.0000
C01249=62.520,106.080,27.030,-0.0500,-0.0400,1.0000
C01250=63.910,103.840,26.920,-0.1000,-0.0500,0.9900
C01251=64.730,101.740,26.710,-0.1700,-0.0600,0.9800
C01252=65.570,99.690,26.420,-0.2600,-0.1200,0.9600
C01253=66.920,97.540,26.130,-0.3200,-0.2300,0.9200
C01254=69.440,94.930,25.900,-0.3100,-0.3400,0.8900
C01255=73.640,91.400,25.810,-0.3100,-0.3700,0.8800
C01256=78.230,87.480,25.810,-0.3200,-0.3600,0.8800
C01257=82.990,82.990,25.810,-0.3400,-0.3400,0.8800
C01258=87.480,78.230,25.810,-0.3600,-0.3200,0.8800
C01259=91.400,73.640,25.810,-0.3700,-0.3100,0.8800
C01260=94.930,69.440,25.900,-0.3400,-0.3100,0.8900
C01261=97.540,66.920,26.130,-0.2300,-0.3200,0.9200
C01262=99.690,65.570,26.420,-0.1200,-0.2600,0.9600
C01263=101.740,64.730,26.710,-0.0600,-0.1700,0.9800
C01264=103.840,63.910,26.920,-0.0500,-0.1000,0.9900
C01265=106.080,62.520,27.030,-0.0400,-0.0500,1.0000
C01266=108.600,60.060,27.080,-0.0200,-0.0200,1.0000
C01267=111.060,56.820,27.120,-0.0000,-0.0000,1.0000
C01268=113.060,53.230,27.170,-0.0000,-0.0000,1.0000
C01269=114.720,49.630,27.200,-0.0000,-0.0000,1.0000
C01270=116.210,46.020,27.200,-0.0000,-0.0000,1.0000
C01271=117.580,42.310,27.170,-0.0000,-0.0000,1.0000
C01272=118.710,38.350,27.120,-0.0000,-0.0000,1.0000
C01273=119.260,34.320,27.080,-0.0300,-0.0000,1.0000
C01274=119.220,30.810,27.030,-0.0700,0.0100,1.0000
C01275=118.620,28.240,26.920,-0.1100,0.0400,0.9900
C01276=117.720,26.170,26.710,-0.1600,0.0800,0.9800
C01277=116.850,24.130,26.420,-0.2700,0.1000,0.9600
C01278=116.290,21.650,26.130,-0.3900,0.0600,0.9200
C01279=116.230,18.030,25.900,-0.4600,-0.0200,0.8900
C01280=116.700,12.560,25.810,-0.4800,-0.0400,0.8800
C01281=117.170,6.540,25.810,-0.4800,-0.0300,0.8800
C01282=117.360,0.000,25.810,-0.4800,0.0000,0.8800
C01283=117.170,-6.540,25.810,-0.4800,0.0300,0.8800
C01284=116.700,-12.560,25.810,-0.4800,0.0400,0.8800
C01285=116.230,-18.030,25.900,-0.4600,0.0200,0.8900
C01286=116.290,-21.650,26.130,-0.3900,-0.0600,0.9200
C01287=116.850,-24.130,26.420,-0.2700,-0.1000,0.9600
C01288=117.720,-26.170,26.710,-0.1600,-0.0800,0.9800
C01289=118.620,-28.240,26.920,-0.1100,-0.0400,0.9900
C01290=119.220,-30.810,27.030,-0.0700,-0.0100,1.0000
C01291=119.260,-34.320,27.080,-0.0300,0.0000,1.0000
C01292=118.710,-38.350,27.120,-0.0000,0.0000,1.0000
C01293=117.580,-42.310,27.170,-0.0000,0.0000,1.0000
C01294=116.210,-46.020,27.200,-0.0000,0.0000,1.0000
C01295=114.720,-49.630,27.200,-0.0000,0.0000,1.0000
C01296=113.060,-53.230,27.170,-0.0000,0.0000,1.0000
C01297=111.060,-56.820,27.120,-0.0000,0.0000,1.0000
C01298=108.600,-60.060,27.080,-0.0200,0.0200,1.0000
C01299=106.080,-62.520,27.030,-0.0400,0.0500,1.0000
C01300=103.840,-63.910,26.920,-0.0500,0.1000,0.9900
C01301=101.740,-64.730,26.710,-0.0600,0.1700,0.9800
C01302=99.690,-65.570,26.420,-0.1200,0.2600,0.9600
C01303=97.540,-66.920,26.130,-0.2300,0.3200,0.9200
C01304=94.930,-69.440,25.900,-0.3400,0.3100,0.8900
C01305=91.400,-73.640,25.810,-0.3700,0.3100,0.8800
C01306=87.480,-78.230,25.810,-0.3600,0.3200,0.8800
C01307=82.990,-82.990,25.810,-0.3400,0.3400,0.8800
C01308=78.230,-87.480,25.810,-0.3200,0.3600,0.8800
C01309=73.640,-91.400,25.810,-0.3100,0.3700,0.8800
C01310=69.440,-94.930,25.900,-0.3100,0.3400,0.8900
C01311=66.920,-97.540,26.130,-0.3200,0.2300,0.9200
C01312=65.570,-99.690,26.420,-0.2600,0.1200,0.9600
C01313=64.730,-101.740,26.710,-0.1700,0.0600,0.9800
C01314=63.910,-103.840,26.920,-0.1000,0.0500,0.9900
C01315=62.520,-106.080,27.030,-0.0500,0.0400,1.0000
C01316=60.060,-108.600,27.080,-0.0200,0.0200,1.0000
C01317=56.820,-111.060,27.120,-0.0000,0.0000,1.0000
C01318=53.230,-113.060,27.170,-0.0000,0.0000,1.0000
C01319=49.630,-114.720,27.200,-0.0000,0.0000,1.0000
C01320=46.020,-116.210,27.200,-0.0000,0.0000,1.0000
C01321=42.310,-117.580,27.170,-0.0000,0.0000,1.0000
C01322=38.350,-118.710,27.120,-0.0000,0.0000,1.0000
C01323=34.320,-119.260,27.080,-0.0000,0.0300,1.0000
C01324=30.810,-119.220,27.030,0.0100,0.0700,1.0000
C01325=28.240,-118.620,26.920,0.0400,0.1100,0.9900
C01326=26.170,-117.720,26.710,0.0800,0.1600,0.9800
C01327=24.130,-116.850,26.420,0.1000,0.2700,0.9600
C01328=21.650,-116.290,26.130,0.0600,0.3900,0.9200
C01329=18.030,-116.230,25.900,-0.0200,0.4600,0.8900
C01330=12.560,-116.700,25.810,-0.0400,0.4800,0.8800
C01331=6.540,-117.170,25.810,-0.0300,0.4800,0.8800
C01332=0.000,-117.360,25.810,0.0000,0.4800,0.8800
C01333=0.000,-117.360,25.810,0.0000,0.4800,0.8800
C01334=-6.540,-117.170,25.810,0.0300,0.4800,0.8800
C01335=-12.560,-116.700,25.810,0.0400,0.4800,0.8800
C01336=-18.030,-116.230,25.900,0.0200,0.4600,0.8900
C01337=-21.650,-116.290,26.130,-0.0600,0.3900,0.9200
C01338=-24.130,-116.850,26.420,-0.1000,0.2700,0.9600
C01339=-26.170,-117.720,26.710,-0.0800,0.1600,0.9800
C01340=-28.240,-118.620,26.920,-0.0400,0.1100,0.9900
C01341=-30.810,-119.220,27.030,-0.0100,0.0700,1.0000
C01342=-34.320,-119.260,27.080,0.0000,0.0300,1.0000
C01343=-38.350,-118.710,27.120,0.0000,0.0000,1.0000
C01344=-42.310,-117.580,27.170,0.0000,0.0000,1.0000
C01345=-46.020,-116.210,27.200,0.0000,0.0000,1.0000
C01346=-49.630,-114.720,27.200,0.0000,0.0000,1.0000
C01347=-53.230,-113.060,27.170,0.0000,0.0000,1.0000
C01348=-56.820,-111.060,27.120,0.0000,0.0000,1.0000
C01349=-60.060,-108.600,27.080,0.0200,0.0200,1.0000
C01350=-62.520,-106.080,27.030,0.0500,0.0400,1.0000
C01351=-63.910,-103.840,26.920,0.1000,0.0500,0.9900
C01352=-64.730,-101.740,26.710,0.1700,0.0600,0.9800
C01353=-65.570,-99.690,26.420,0.2600,0.1200,0.9600
C01354=-66.920,-97.540,26.130,0.3200,0.2300,0.9200
C01355=-69.440,-94.930,25.900,0.3100,0.3400,0.8900
C01356=-73.640,-91.400,25.810,0.3100,0.3700,0.8800
C01357=-78.230,-87.480,25.810,0.3200,0.3600,0.8800
C01358=-82.990,-82.990,25.810,0.3400,0.3400,0.8800
C01359=-87.480,-78.230,25.810,0.3600,0.3200,0.8800
C01360=-91.400,-73.640,25.810,0.3700,0.3100,0.8800
C01361=-94.930,-69.440,25.900,0.3400,0.3100,0.8900
C01362=-97.540,-66.920,26.130,0.2300,0.3200,0.9200
C01363=-99.690,-65.570,26.420,0.1200,0.2600,0.9600
C01364=-101.740,-64.730,26.710,0.0600,0.1700,0.9800
C01365=-103.840,-63.910,26.920,0.0500,0.1000,0.9900
C01366=-106.080,-62.520,27.030,0.0400,0.0500,1.0000
C01367=-108.600,-60.060,27.080,0.0200,0.0200,1.0000
C01368=-111.060,-56.820,27.120,0.0000,0.0000,1.0000
C01369=-113.060,-53.230,27.170,0.0000,0.0000,1.0000
C01370=-114.720,-49.630,27.200,0.0000,0.0000,1.0000
C01371=-116.210,-46.020,27.200,0.0000,0.0000,1.0000
C01372=-117.580,-42.310,27.170,0.0000,0.0000,1.0000
C01373=-118.710,-38.350,27.120,0.0000,0.0000,1.0000
C01374=-119.260,-34.320,27.080,0.0300,0.0000,1.0000
C01375=-119.220,-30.810,27.030,0.0700,-0.0100,1.0000
C01376=-118.620,-28.240,26.920,0.1100,-0.0400,0.9900
C01377=-117.720,-26.170,26.710,0.1600,-0.0800,0.9800
C01378=-116.850,-24.130,26.420,0.2700,-0.1000,0.9600
C01379=-116.290,-21.650,26.130,0.3900,-0.0600,0.9200
C01380=-116.230,-18.030,25.900,0.4600,0.0200,0.8900
C01381=-116.700,-12.560,25.810,0.4800,0.0400,0.8800
C01382=-117.170,-6.540,25.810,0.4800,0.0300,0.8800
C01383=-117.360,0.000,25.810,0.4800,-0.0000,0.8800
C01384=-117.170,6.540,25.810,0.4800,-0.0300,0.8800
C01385=-116.700,12.560,25.810,0.4800,-0.0400,0.8800
C01386=-116.230,18.030,25.900,0.4600,-0.0200,0.8900
C01387=-116.290,21.650,26.130,0.3900,0.0600,0.9200
C01388=-116.850,24.130,26.420,0.2700,0.1000,0.9600
C01389=-117.720,26.170,26.710,0.1600,0.0800,0.9800
C01390=-118.620,28.240,26.920,0.1100,0.0400,0.9900
C01391=-119.220,30.810,27.030,0.0700,0.0100,1.0000
C01392=-119.260,34.320,27.080,0.0300,-0.0000,1.0000
C01393=-118.710,38.350,27.120,0.0000,-0.0000,1.0000
C01394=-117.580,42.310,27.170,0.0000,-0.0000,1.0000
C01395=-116.210,46.020,27.200,0.0000,-0.0000,1.0000
C01396=-114.720,49.630,27.200,0.0000,-0.0000,1.0000
C01397=-113.060,53.230,27.170,0.0000,-0.0000,1.0000
C01398=-111.060,56.820,27.120,0.0000,-0.0000,1.0000
C01399=-108.600,60.060,27.080,0.0200,-0.0200,1.0000
C01400=-106.080,62.520,27.030,0.0400,-0.0500,1.0000
C01401=-103.840,63.910,26.920,0.0500,-0.1000,0.9900
C01402=-101.740,64.730,26.710,0.0600,-0.1700,0.9800
C01403=-99.690,65.570,26.420,0.1200,-0.2600,0.9600
C01404=-97.540,66.920,26.130,0.2300,-0.3200,0.9200
C01405=-94.930,69.440,25.900,0.3400,-0.3100,0.8900
C01406=-91.400,73.640,25.810,0.3700,-0.3100,0.8800
C01407=-87.480,78.230,25.810,0.3600,-0.3200,0.8800
C01408=-82.990,82.990,25.810,0.3400,-0.3400,0.8800
C01409=-78.230,87.480,25.810,0.3200,-0.3600,0.8800
C01410=-73.640,91.400,25.810,0.3100,-0.3700,0.8800
C01411=-69.440,94.930,25.900,0.3100,-0.3400,0.8900
C01412=-66.920,97.540,26.130,0.3200,-0.2300,0.9200
C01413=-65.570,99.690,26.420,0.2600,-0.1200,0.9600
C01414=-64.730,101.740,26.710,0.1700,-0.0600,0.9800
C01415=-63.910,103.840,26.920,0.1000,-0.0500,0.9900
C01416=-62.520,106.080,27.030,0.0500,-0.0400,1.0000
C01417=-60.060,108.600,27.080,0.0200,-0.0200,1.0000
C01418=-56.820,111.060,27.120,0.0000,-0.0000,1.0000
C01419=-53.230,113.060,27.170,0.0000,-0.0000,1.0000
C01420=-49.630,114.720,27.200,0.0000,-0.0000,1.0000
C01421=-46.020,116.210,27.200,0.0000,-0.0000,1.0000
C01422=-42.310,117.580,27.170,0.0000,-0.0000,1.0000
C01423=-38.350,118.710,27.120,0.0000,-0.0000,1.0000
C01424=-34.320,119.260,27.080,0.0000,-0.0300,1.0000
C01425=-30.810,119.220,27.030,-0.0100,-0.0700,1.0000
C01426=-28.240,118.620,26.920,-0.0400,-0.1100,0.9900
C01427=-26.170,117.720,26.710,-0.0800,-0.1600,0.9800
C01428=-24.130,116.850,26.420,-0.1000,-0.2700,0.9600
C01429=-21.650,116.290,26.130,-0.0600,-0.3900,0.9200
C01430=-18.030,116.230,25.900,0.0200,-0.4600,0.8900
C01431=-12.560,116.700,25.810,0.0400,-0.4800,0.8800
C01432=-6.540,117.170,25.810,0.0300,-0.4800,0.8800
C01433=0.000,117.360,25.810,0.0000,-0.4800,0.8800
C01434=0.000,116.530,27.290,0.0000,-0.4900,0.8700
C01435=-6.470,116.350,27.290,0.0300,-0.4900,0.8700
C01436=-12.430,115.880,27.300,0.0400,-0.4900,0.8700
C01437=-17.870,115.440,27.400,0.0100,-0.4700,0.8800
C01438=-21.460,115.580,27.660,-0.0800,-0.4000,0.9100
C01439=-23.910,116.250,28.000,-0.1200,-0.2600,0.9600
C01440=-25.930,117.260,28.330,-0.0900,-0.1500,0.9900
C01441=-27.990,118.320,28.580,-0.0400,-0.1000,0.9900
C01442=-30.530,119.070,28.700,-0.0100,-0.0600,1.0000
C01443=-34.060,119.230,28.760,0.0000,-0.0300,1.0000
C01444=-38.140,118.750,28.810,0.0000,-0.0000,1.0000
C01445=-42.180,117.630,28.860,0.0000,-0.0000,1.0000
C01446=-45.980,116.230,28.900,0.0000,-0.0000,1.0000
C01447=-49.680,114.700,28.900,0.0000,-0.0000,1.0000
C01448=-53.350,113.000,28.860,0.0000,-0.0000,1.0000
C01449=-56.990,110.940,28.810,0.0000,-0.0000,1.0000
C01450=-60.220,108.400,28.760,0.0200,-0.0200,1.0000
C01451=-62.600,105.780,28.700,0.0500,-0.0400,1.0000
C01452=-63.870,103.450,28.580,0.1000,-0.0400,0.9900
C01453=-64.580,101.250,28.330,0.1700,-0.0400,0.9900
C01454=-65.290,99.110,28.000,0.2700,-0.1000,0.9600
C01455=-66.550,96.900,27.660,0.3400,-0.2200,0.9100
C01456=-68.990,94.270,27.400,0.3300,-0.3400,0.8800
C01457=-73.150,90.730,27.300,0.3200,-0.3800,0.8700
C01458=-77.700,86.840,27.290,0.3300,-0.3700,0.8700
C01459=-82.400,82.400,27.290,0.3500,-0.3500,0.8700
C01460=-86.840,77.700,27.290,0.3700,-0.3300,0.8700
C01461=-90.730,73.150,27.300,0.3800,-0.3200,0.8700
C01462=-94.270,68.990,27.400,0.3400,-0.3300,0.8800
C01463=-96.900,66.550,27.660,0.2200,-0.3400,0.9100
C01464=-99.110,65.290,28.000,0.1000,-0.2700,0.9600
C01465=-101.250,64.580,28.330,0.0400,-0.1700,0.9900
C01466=-103.450,63.870,28.580,0.0400,-0.1000,0.9900
C01467=-105.780,62.600,28.700,0.0400,-0.0500,1.0000
C01468=-108.400,60.220,28.760,0.0200,-0.0200,1.0000
C01469=-110.940,56.990,28.810,0.0000,-0.0000,1.0000
C01470=-113.000,53.350,28.860,0.0000,-0.0000,1.0000
C01471=-114.700,49.680,28.900,0.0000,-0.0000,1.0000
C01472=-116.230,45.980,28.900,0.0000,-0.0000,1.0000
C01473=-117.630,42.180,28.860,0.0000,-0.0000,1.0000
C01474=-118.750,38.140,28.810,0.0000,-0.0000,1.0000
C01475=-119.230,34.060,28.760,0.0300,-0.0000,1.0000
C01476=-119.070,30.530,28.700,0.0600,0.0100,1.0000
C01477=-118.320,27.990,28.580,0.1000,0.0400,0.9900
C01478=-117.260,25.930,28.330,0.1500,0.0900,0.9900
C01479=-116.250,23.910,28.000,0.2600,0.1200,0.9600
C01480=-115.580,21.460,27.660,0.4000,0.0800,0.9100
C01481=-115.440,17.870,27.400,0.4700,-0.0100,0.8800
C01482=-115.880,12.430,27.300,0.4900,-0.0400,0.8700
C01483=-116.350,6.470,27.290,0.4900,-0.0300,0.8700
C01484=-116.530,0.000,27.290,0.4900,-0.0000,0.8700
C01485=-116.350,-6.470,27.290,0.4900,0.0300,0.8700
C01486=-115.880,-12.430,27.300,0.4900,0.0400,0.8700
C01487=-115.440,-17.870,27.400,0.4700,0.0100,0.8800
C01488=-115.580,-21.460,27.660,0.4000,-0.0800,0.9100
C01489=-116.250,-23.910,28.000,0.2600,-0.1200,0.9600
C01490=-117.260,-25.930,28.330,0.1500,-0.0900,0.9900
C01491=-118.320,-27.990,28.580,0.1000,-0.0400,0.9900
C01492=-119.070,-30.530,28.700,0.0600,-0.0100,1.0000
C01493=-119.230,-34.060,28.760,0.0300,0.0000,1.0000
C01494=-118.750,-38.140,28.810,0.0000,0.0000,1.0000
C01495=-117.630,-42.180,28.860,0.0000,0.0000,1.0000
C01496=-116.230,-45.980,28.900,0.0000,0.0000,1.0000
C01497=-114.700,-49.680,28.900,0.0000,0.0000,1.0000
C01498=-113.000,-53.350,28.860,0.0000,0.0000,1.0000
C01499=-110.940,-56.990,28.810,0.0000,0.0000,1.0000
C01500=-108.400,-60.220,28.760,0.0200,0.0200,1.0000
C01501=-105.780,-62.600,28.700,0.0400,0.0500,1.0000
C01502=-103.450,-63.870,28.580,0.0400,0.1000,0.9900
C01503=-101.250,-64.580,28.330,0.0400,0.1700,0.9900
C01504=-99.110,-65.290,28.000,0.1000,0.2700,0.9600
C01505=-96.900,-66.550,27.660,0.2200,0.3400,0.9100
C01506=-94.270,-68.990,27.400,0.3400,0.3300,0.8800
C01507=-90.730,-73.150,27.300,0.3800,0.3200,0.8700
C01508=-86.840,-77.700,27.290,0.3700,0.3300,0.8700
C01509=-82.400,-82.400,27.290,0.3500,0.3500,0.8700
C01510=-77.700,-86.840,27.290,0.3300,0.3700,0.8700
C01511=-73.150,-90.730,27.300,0.3200,0.3800,0.8700
C01512=-68.990,-94.270,27.400,0.3300,0.3400,0.8800
C01513=-66.550,-96.900,27.660,0.3400,0.2200,0.9100
C01514=-65.290,-99.110,28.000,0.2700,0.1000,0.9600
C01515=-64.580,-101.250,28.330,0.1700,0.0400,0.9900
C01516=-63.870,-103.450,28.580,0.1000,0.0400,0.9900
C01517=-62.600,-105.780,28.700,0.0500,0.0400,1.0000
C01518=-60.220,-108.400,28.760,0.0200,0.0200,1.0000
C01519=-56.990,-110.940,28.810,0.0000,0.0000,1.0000
C01520=-53.350,-113.000,28.860,0.0000,0.0000,1.0000
C01521=-49.680,-114.700,28.900,0.0000,0.0000,1.0000
C01522=-45.980,-116.230,28.900,0.0000,0.0000,1.0000
C01523=-42.180,-117.630,28.860,0.0000,0.0000,1.0000
C01524=-38.140,-118.750,28.810,0.0000,0.0000,1.0000
C01525=-34.060,-119.230,28.760,0.0000,0.0300,1.0000
C01526=-30.530,-119.070,28.700,-0.0100,0.0600,1.0000
C01527=-27.990,-118.320,28.580,-0.0400,0.1000,0.9900
C01528=-25.930,-117.260,28.330,-0.0900,0.1500,0.9900
C01529=-23.910,-116.250,28.000,-0.1200,0.2600,0.9600
C01530=-21.460,-115.580,27.660,-0.0800,0.4000,0.9100
C01531=-17.870,-115.440,27.400,0.0100,0.4700,0.8800
C01532=-12.430,-115.880,27.300,0.0400,0.4900,0.8700
C01533=-6.470,-116.350,27.290,0.0300,0.4900,0.8700
C01534=0.000,-116.530,27.290,0.0000,0.4900,0.8700
C01535=0.000,-116.530,27.290,0.0000,0.4900,0.8700
C01536=6.470,-116.350,27.290,-0.0300,0.4900,0.8700
C01537=12.430,-115.880,27.300,-0.0400,0.4900,0.8700
C01538=17.870,-115.440,27.400,-0.0100,0.4700,0.8800
C01539=21.460,-115.580,27.660,0.0800,0.4000,0.9100
C01540=23.910,-116.250,28.000,0.1200,0.2600,0.9600
C01541=25.930,-117.260,28.330,0.0900,0.1500,0.9900
C01542=27.990,-118.320,28.580,0.0400,0.1000,0.9900
C01543=30.530,-119.070,28.700,0.0100,0.0600,1.0000
C01544=34.060,-119.230,28.760,-0.0000,0.0300,1.0000
C01545=38.140,-118.750,28.810,-0.0000,0.0000,1.0000
C01546=42.180,-117.630,28.860,-0.0000,0.0000,1.0000
C01547=45.980,-116.230,28.900,-0.0000,0.0000,1.0000
C01548=49.680,-114.700,28.900,-0.0000,0.0000,1.0000
C01549=53.350,-113.000,28.860,-0.0000,0.0000,1.0000
C01550=56.990,-110.940,28.810,-0.0000,0.0000,1.0000
C01551=60.220,-108.400,28.760,-0.0200,0.0200,1.0000
C01552=62.600,-105.780,28.700,-0.0500,0.0400,1.0000
C01553=63.870,-103.450,28.580,-0.1000,0.0400,0.9900
C01554=64.580,-101.250,28.330,-0.1700,0.0400,0.9900
C01555=65.290,-99.110,28.000,-0.2700,0.1000,0.9600
C01556=66.550,-96.900,27.660,-0.3400,0.2200,0.9100
C01557=68.990,-94.270,27.400,-0.3300,0.3400,0.8800
C01558=73.150,-90.730,27.300,-0.3200,0.3800,0.8700
C01559=77.700,-86.840,27.290,-0.3300,0.3700,0.8700
C01560=82.400,-82.400,27.290,-0.3500,0.3500,0.8700
C01561=86.840,-77.700,27.290,-0.3700,0.3300,0.8700
C01562=90.730,-73.150,27.300,-0.3800,0.3200,0.8700
C01563=94.270,-68.990,27.400,-0.3400,0.3300,0.8800
C01564=96.900,-66.550,27.660,-0.2200,0.3400,0.9100
C01565=99.110,-65.290,28.000,-0.1000,0.2700,0.9600
C01566=101.250,-64.580,28.330,-0.0400,0.1700,0.9900
C01567=103.450,-63.870,28.580,-0.0400,0.1000,0.9900
C01568=105.780,-62.600,28.700,-0.0400,0.0500,1.0000
C01569=108.400,-60.220,28.760,-0.0200,0.0200,1.0000
C01570=110.940,-56.990,28.810,-0.0000,0.0000,1.0000
C01571=113.000,-53.350,28.860,-0.0000,0.0000,1.0000
C01572=114.700,-49.680,28.900,-0.0000,0.0000,1.0000
C01573=116.230,-45.980,28.900,-0.0000,0.0000,1.0000
C01574=117.630,-42.180,28.860,-0.0000,0.0000,1.0000
C01575=118.750,-38.140,28.810,-0.0000,0.0000,1.0000
C01576=119.230,-34.060,28.760,-0.0300,0.0000,1.0000
C01577=119.070,-30.530,28.700,-0.0600,-0.0100,1.0000
C01578=118.320,-27.990,28.580,-0.1000,-0.0400,0.9900
C01579=117.260,-25.930,28.330,-0.1500,-0.0900,0.9900
C01580=116.250,-23.910,28.000,-0.2600,-0.1200,0.9600
C01581=115.580,-21.460,27.660,-0.4000,-0.0800,0.9100
C01582=115.440,-17.870,27.400,-0.4700,0.0100,0.8800
C01583=115.880,-12.430,27.300,-0.4900,0.0400,0.8700
C01584=116.350,-6.470,27.290,-0.4900,0.0300,0.8700
C01585=116.530,0.000,27.290,-0.4900,0.0000,0.8700
C01586=116.350,6.470,27.290,-0.4900,-0.0300,0.8700
C01587=115.880,12.430,27.300,-0.4900,-0.0400,0.8700
C01588=115.440,17.870,27.400,-0.4700,-0.0100,0.8800
C01589=115.580,21.460,27.660,-0.4000,0.0800,0.9100
C01590=116.250,23.910,28.000,-0.2600,0.1200,0.9600
C01591=117.260,25.930,28.330,-0.1500,0.0900,0.9900
C01592=118.320,27.990,28.580,-0.1000,0.0400,0.9900
C01593=119.070,30.530,28.700,-0.0600,0.0100,1.0000
C01594=119.230,34.060,28.760,-0.0300,-0.0000,1.0000
C01595=118.750,38.140,28.810,-0.0000,-0.0000,1.0000
C01596=117.630,42.180,28.860,-0.0000,-0.0000,1.0000
C01597=116.230,45.980,28.900,-0.0000,-0.0000,1.0000
C01598=114.700,49.680,28.900,-0.0000,-0.0000,1.0000
C01599=113.000,53.350,28.860,-0.0000,-0.0000,1.0000
C01600=110.940,56.990,28.810,-0.0000,-0.0000,1.0000
C01601=108.400,60.220,28.760,-0.0200,-0.0200,1.0000
C01602=105.780,62.600,28.700,-0.0400,-0.0500,1.0000
C01603=103.450,63.870,28.580,-0.0400,-0.1000,0.9900
C01604=101.250,64.580,28.330,-0.0400,-0.1700,0.9900
C01605=99.110,65.290,28.000,-0.1000,-0.2700,0.9600
C01606=96.900,66.550,27.660,-0.2200,-0.3400,0.9100
C01607=94.270,68.990,27.400,-0.3400,-0.3300,0.8800
C01608=90.730,73.150,27.300,-0.3800,-0.3200,0.8700
C01609=86.840,77.700,27.290,-0.3700,-0.3300,0.8700
C01610=82.400,82.400,27.290,-0.3500,-0.3500,0.8700
C01611=77.700,86.840,27.290,-0.3300,-0.3700,0.8700
C01612=73.150,90.730,27.300,-0.3200,-0.3800,0.8700
C01613=68.990,94.270,27.400,-0.3300,-0.3400,0.8800
C01614=66.550,96.900,27.660,-0.3400,-0.2200,0.9100
C01615=65.290,99.110,28.000,-0.2700,-0.1000,0.9600
C01616=64.580,101.250,28.330,-0.1700,-0.0400,0.9900
C01617=63.870,103.450,28.580,-0.1000,-0.0400,0.9900
C01618=62.600,105.780,28.700,-0.0500,-0.0400,1.0000
C01619=60.220,108.400,28.760,-0.0200,-0.0200,1.0000
C01620=56.990,110.940,28.810,-0.0000,-0.0000,1.0000
C01621=53.350,113.000,28.860,-0.0000,-0.0000,1.0000
C01622=49.680,114.700,28.900,-0.0000,-0.0000,1.0000
C01623=45.980,116.230,28.900,-0.0000,-0.0000,1.0000
C01624=42.180,117.630,28.860,-0.0000,-0.0000,1.0000
C01625=38.140,118.750,28.810,-0.0000,-0.0000,1.0000
C01626=34.060,119.230,28.760,-0.0000,-0.0300,1.0000
C01627=30.530,119.070,28.700,0.0100,-0.0600,1.0000
C01628=27.990,118.320,28.580,0.0400,-0.1000,0.9900
C01629=25.930,117.260,28.330,0.0900,-0.1500,0.9900
C01630=23.910,116.250,28.000,0.1200,-0.2600,0.9600
C01631=21.460,115.580,27.660,0.0800,-0.4000,0.9100
C01632=17.870,115.440,27.400,-0.0100,-0.4700,0.8800
C01633=12.430,115.880,27.300,-0.0400,-0.4900,0.8700
C01634=6.470,116.350,27.290,-0.0300,-0.4900,0.8700
C01635=0.000,116.530,27.290,0.0000,-0.4900,0.8700
C01636=0.000,115.680,28.760,0.0000,-0.5100,0.8600
C01637=6.390,115.500,28.760,-0.0300,-0.5100,0.8600
C01638=12.300,115.040,28.770,-0.0400,-0.5100,0.8600
C01639=17.710,114.630,28.880,-0.0100,-0.4900,0.8700
C01640=21.260,114.840,29.170,0.1000,-0.4000,0.9100
C01641=23.690,115.630,29.560,0.1300,-0.2400,0.9600
C01642=25.690,116.780,29.940,0.0900,-0.1300,0.9900
C01643=27.720,118.000,30.230,0.0400,-0.0800,1.0000
C01644=30.250,118.910,30.370,0.0100,-0.0600,1.0000
C01645=33.800,119.200,30.440,-0.0000,-0.0200,1.0000
C01646=37.930,118.790,30.500,-0.0000,-0.0000,1.0000
C01647=42.040,117.670,30.560,-0.0000,-0.0000,1.0000
C01648=45.930,116.250,30.590,-0.0000,-0.0000,1.0000
C01649=49.720,114.680,30.590,-0.0000,-0.0000,1.0000
C01650=53.480,112.940,30.560,-0.0000,-0.0000,1.0000
C01651=57.170,110.810,30.500,-0.0000,-0.0000,1.0000
C01652=60.390,108.190,30.440,-0.0200,-0.0200,1.0000
C01653=62.700,105.470,30.370,-0.0500,-0.0300,1.0000
C01654=63.840,103.050,30.230,-0.0900,-0.0300,1.0000
C01655=64.410,100.740,29.940,-0.1600,-0.0300,0.9900
C01656=65.010,98.510,29.560,-0.2700,-0.0800,0.9600
C01657=66.170,96.240,29.170,-0.3500,-0.2100,0.9100
C01658=68.530,93.580,28.880,-0.3400,-0.3500,0.8700
C01659=72.640,90.040,28.770,-0.3300,-0.3900,0.8600
C01660=77.150,86.190,28.760,-0.3400,-0.3800,0.8600
C01661=81.800,81.800,28.760,-0.3600,-0.3600,0.8600
C01662=86.190,77.150,28.760,-0.3800,-0.3400,0.8600
C01663=90.040,72.640,28.770,-0.3900,-0.3300,0.8600
C01664=93.580,68.530,28.880,-0.3500,-0.3400,0.8700
C01665=96.240,66.170,29.170,-0.2100,-0.3500,0.9100
C01666=98.510,65.010,29.560,-0.0800,-0.2700,0.9600
C01667=100.740,64.410,29.940,-0.0300,-0.1600,0.9900
C01668=103.050,63.840,30.230,-0.0300,-0.0900,1.0000
C01669=105.470,62.700,30.370,-0.0300,-0.0500,1.0000
C01670=108.190,60.390,30.440,-0.0200,-0.0200,1.0000
C01671=110.810,57.170,30.500,-0.0000,-0.0000,1.0000
C01672=112.940,53.480,30.560,-0.0000,-0.0000,1.0000
C01673=114.680,49.720,30.590,-0.0000,-0.0000,1.0000
C01674=116.250,45.930,30.590,-0.0000,-0.0000,1.0000
C01675=117.670,42.040,30.560,-0.0000,-0.0000,1.0000
C01676=118.790,37.930,30.500,-0.0000,-0.0000,1.0000
C01677=119.200,33.800,30.440,-0.0200,-0.0000,1.0000
C01678=118.910,30.250,30.370,-0.0600,0.0100,1.0000
C01679=118.000,27.720,30.230,-0.0800,0.0400,1.0000
C01680=116.780,25.690,29.940,-0.1300,0.0900,0.9900
C01681=115.630,23.690,29.560,-0.2400,0.1300,0.9600
C01682=114.840,21.260,29.170,-0.4000,0.1000,0.9100
C01683=114.630,17.710,28.880,-0.4900,-0.0100,0.8700
C01684=115.040,12.300,28.770,-0.5100,-0.0400,0.8600
C01685=115.500,6.390,28.760,-0.5100,-0.0300,0.8600
C01686=115.680,0.000,28.760,-0.5100,0.0000,0.8600
C01687=115.500,-6.390,28.760,-0.5100,0.0300,0.8600
C01688=115.040,-12.300,28.770,-0.5100,0.0400,0.8600
C01689=114.630,-17.710,28.880,-0.4900,0.0100,0.8700
C01690=114.840,-21.260,29.170,-0.4000,-0.1000,0.9100
C01691=115.630,-23.690,29.560,-0.2400,-0.1300,0.9600
C01692=116.780,-25.690,29.940,-0.1300,-0.0900,0.9900
C01693=118.000,-27.720,30.230,-0.0800,-0.0400,1.0000
C01694=118.910,-30.250,30.370,-0.0600,-0.0100,1.0000
C01695=119.200,-33.800,30.440,-0.0200,0.0000,1.0000
C01696=118.790,-37.930,30.500,-0.0000,0.0000,1.0000
C01697=117.670,-42.040,30.560,-0.0000,0.0000,1.0000
C01698=116.250,-45.930,30.590,-0.0000,0.0000,1.0000
C01699=114.680,-49.720,30.590,-0.0000,0.0000,1.0000
C01700=112.940,-53.480,30.560,-0.0000,0.0000,1.0000
C01701=110.810,-57.170,30.500,-0.0000,0.0000,1.0000
C01702=108.190,-60.390,30.440,-0.0200,0.0200,1.0000
C01703=105.470,-62.700,30.370,-0.0300,0.0500,1.0000
C01704=103.050,-63.840,30.230,-0.0300,0.0900,1.0000
C01705=100.740,-64.410,29.940,-0.0300,0.1600,0.9900
C01706=98.510,-65.010,29.560,-0.0800,0.2700,0.9600
C01707=96.240,-66.170,29.170,-0.2100,0.3500,0.9100
C01708=93.580,-68.530,28.880,-0.3500,0.3400,0.8700
C01709=90.040,-72.640,28.770,-0.3900,0.3300,0.8600
C01710=86.190,-77.150,28.760,-0.3800,0.3400,0.8600
C01711=81.800,-81.800,28.760,-0.3600,0.3600,0.8600
C01712=77.150,-86.190,28.760,-0.3400,0.3800,0.8600
C01713=72.640,-90.040,28.770,-0.3300,0.3900,0.8600
C01714=68.530,-93.580,28.880,-0.3400,0.3500,0.8700
C01715=66.170,-96.240,29.170,-0.3500,0.2100,0.9100
C01716=65.010,-98.510,29.560,-0.2700,0.0800,0.9600
C01717=64.410,-100.740,29.940,-0.1600,0.0300,0.9900
C01718=63.840,-103.050,30.230,-0.0900,0.0300,1.0000
C01719=62.700,-105.470,30.370,-0.0500,0.0300,1.0000
C01720=60.390,-108.190,30.440,-0.0200,0.0200,1.0000
C01721=57.170,-110.810,30.500,-0.0000,0.0000,1.0000
C01722=53.480,-112.940,30.560,-0.0000,0.0000,1.0000
C01723=49.720,-114.680,30.590,-0.0000,0.0000,1.0000
C01724=45.930,-116.250,30.590,-0.0000,0.0000,1.0000
C01725=42.040,-117.670,30.560,-0.0000,0.0000,1.0000
C01726=37.930,-118.790,30.500,-0.0000,0.0000,1.0000
C01727=33.800,-119.200,30.440,-0.0000,0.0200,1.0000
C01728=30.250,-118.910,30.370,0.0100,0.0600,1.0000
C01729=27.720,-118.000,30.230,0.0400,0.0800,1.0000
C01730=25.690,-116.780,29.940,0.0900,0.1300,0.9900
C01731=23.690,-115.630,29.560,0.1300,0.2400,0.9600
C01732=21.260,-114.840,29.170,0.1000,0.4000,0.9100
C01733=17.710,-114.630,28.880,-0.0100,0.4900,0.8700
C01734=12.300,-115.040,28.770,-0.0400,0.5100,0.8600
C01735=6.390,-115.500,28.760,-0.0300,0.5100,0.8600
C01736=0.000,-115.680,28.760,0.0000,0.5100,0.8600
C01737=0.000,-115.680,28.760,0.0000,0.5100,0.8600
C01738=-6.390,-115.500,28.760,0.0300,0.5100,0.8600
C01739=-12.300,-115.040,28.770,0.0400,0.5100,0.8600
C01740=-17.710,-114.630,28.880,0.0100,0.4900,0.8700
C01741=-21.260,-114.840,29.170,-0.1000,0.4000,0.9100
C01742=-23.690,-115.630,29.560,-0.1300,0.2400,0.9600
C01743=-25.690,-116.780,29.940,-0.0900,0.1300,0.9900
C01744=-27.720,-118.000,30.230,-0.0400,0.0800,1.0000
C01745=-30.250,-118.910,30.370,-0.0100,0.0600,1.0000
C01746=-33.800,-119.200,30.440,0.0000,0.0200,1.0000
C01747=-37.930,-118.790,30.500,0.0000,0.0000,1.0000
C01748=-42.040,-117.670,30.560,0.0000,0.0000,1.0000
C01749=-45.930,-116.250,30.590,0.0000,0.0000,1.0000
C01750=-49.720,-114.680,30.590,0.0000,0.0000,1.0000
C01751=-53.480,-112.940,30.560,0.0000,0.0000,1.0000
C01752=-57.170,-110.810,30.500,0.0000,0.0000,1.0000
C01753=-60.390,-108.190,30.440,0.0200,0.0200,1.0000
C01754=-62.700,-105.470,30.370,0.0500,0.0300,1.0000
C01755=-63.840,-103.050,30.230,0.0900,0.0300,1.0000
C01756=-64.410,-100.740,29.940,0.1600,0.0300,0.9900
C01757=-65.010,-98.510,29.560,0.2700,0.0800,0.9600
C01758=-66.170,-96.240,29.170,0.3500,0.2100,0.9100
C01759=-68.530,-93.580,28.880,0.3400,0.3500,0.8700
C01760=-72.640,-90.040,28.770,0.3300,0.3900,0.8600
C01761=-77.150,-86.190,28.760,0.3400,0.3800,0.8600
C01762=-81.800,-81.800,28.760,0.3600,0.3600,0.8600
C01763=-86.190,-77.150,28.760,0.3800,0.3400,0.8600
C01764=-90.040,-72.640,28.770,0.3900,0.3300,0.8600
C01765=-93.580,-68.530,28.880,0.3500,0.3400,0.8700
C01766=-96.240,-66.170,29.170,0.2100,0.3500,0.9100
C01767=-98.510,-65.010,29.560,0.0800,0.2700,0.9600
C01768=-100.740,-64.410,29.940,0.0300,0.1600,0.9900
C01769=-103.050,-63.840,30.230,0.0300,0.0900,1.0000
C01770=-105.470,-62.700,30.370,0.0300,0.0500,1.0000
C01771=-108.190,-60.390,30.440,0.0200,0.0200,1.0000
C01772=-110.810,-57.170,30.500,0.0000,0.0000,1.0000
C01773=-112.940,-53.480,30.560,0.0000,0.0000,1.0000
C01774=-114.680,-49.720,30.590,0.0000,0.0000,1.0000
C01775=-116.250,-45.930,30.590,0.0000,0.0000,1.0000
C01776=-117.670,-42.040,30.560,0.0000,0.0000,1.0000
C01777=-118.790,-37.930,30.500,0.0000,0.0000,1.0000
C01778=-119.200,-33.800,30.440,0.0200,0.0000,1.0000
C01779=-118.910,-30.250,30.370,0.0600,-0.0100,1.0000
C01780=-118.000,-27.720,30.230,0.0800,-0.0400,1.0000
C01781=-116.780,-25.690,29.940,0.1300,-0.0900,0.9900
C01782=-115.630,-23.690,29.560,0.2400,-0.1300,0.9600
C01783=-114.840,-21.260,29.170,0.4000,-0.1000,0.9100
C01784=-114.630,-17.710,28.880,0.4900,0.0100,0.8700
C01785=-115.040,-12.300,28.770,0.5100,0.0400,0.8600
C01786=-115.500,-6.390,28.760,0.5100,0.0300,0.8600
C01787=-115.680,0.000,28.760,0.5100,-0.0000,0.8600
C01788=-115.500,6.390,28.760,0.5100,-0.0300,0.8600
C01789=-115.040,12.300,28.770,0.5100,-0.0400,0.8600
C01790=-114.630,17.710,28.880,0.4900,-0.0100,0.8700
C01791=-114.840,21.260,29.170,0.4000,0.1000,0.9100
C01792=-115.630,23.690,29.560,0.2400,0.1300,0.9600
C01793=-116.780,25.690,29.940,0.1300,0.0900,0.9900
C01794=-118.000,27.720,30.230,0.0800,0.0400,1.0000
C01795=-118.910,30.250,30.370,0.0600,0.0100,1.0000
C01796=-119.200,33.800,30.440,0.0200,-0.0000,1.0000
C01797=-118.790,37.930,30.500,0.0000,-0.0000,1.0000
C01798=-117.670,42.040,30.560,0.0000,-0.0000,1.0000
C01799=-116.250,45.930,30.590,0.0000,-0.0000,1.0000
C01800=-114.680,49.720,30.590,0.0000,-0.0000,1.0000
C01801=-112.940,53.480,30.560,0.0000,-0.0000,1.0000
C01802=-110.810,57.170,30.500,0.0000,-0.0000,1.0000
C01803=-108.190,60.390,30.440,0.0200,-0.0200,1.0000
C01804=-105.470,62.700,30.370,0.0300,-0.0500,1.0000
C01805=-103.050,63.840,30.230,0.0300,-0.0900,1.0000
C01806=-100.740,64.410,29.940,0.0300,-0.1600,0.9900
C01807=-98.510,65.010,29.560,0.0800,-0.2700,0.9600
C01808=-96.240,66.170,29.170,0.2100,-0.3500,0.9100
C01809=-93.580,68.530,28.880,0.3500,-0.3400,0.8700
C01810=-90.040,72.640,28.770,0.3900,-0.3300,0.8600
C01811=-86.190,77.150,28.760,0.3800,-0.3400,0.8600
C01812=-81.800,81.800,28.760,0.3600,-0.3600,0.8600
C01813=-77.150,86.190,28.760,0.3400,-0.3800,0.8600
C01814=-72.640,90.040,28.770,0.3300,-0.3900,0.8600
C01815=-68.530,93.580,28.880,0.3400,-0.3500,0.8700
C01816=-66.170,96.240,29.170,0.3500,-0.2100,0.9100
C01817=-65.010,98.510,29.560,0.2700,-0.0800,0.9600
C01818=-64.410,100.740,29.940,0.1600,-0.0300,0.9900
C01819=-63.840,103.050,30.230,0.0900,-0.0300,1.0000
C01820=-62.700,105.470,30.370,0.0500,-0.0300,1.0000
C01821=-60.390,108.190,30.440,0.0200,-0.0200,1.0000
C01822=-57.170,110.810,30.500,0.0000,-0.0000,1.0000
C01823=-53.480,112.940,30.560,0.0000,-0.0000,1.0000
C01824=-49.720,114.680,30.590,0.0000,-0.0000,1.0000
C01825=-45.930,116.250,30.590,0.0000,-0.0000,1.0000
C01826=-42.040,117.670,30.560,0.0000,-0.0000,1.0000
C01827=-37.930,118.790,30.500,0.0000,-0.0000,1.0000
C01828=-33.800,119.200,30.440,0.0000,-0.0200,1.0000
C01829=-30.250,118.910,30.370,-0.0100,-0.0600,1.0000
C01830=-27.720,118.000,30.230,-0.0400,-0.0800,1.0000
C01831=-25.690,116.780,29.940,-0.0900,-0.1300,0.9900
C01832=-23.690,115.630,29.560,-0.1300,-0.2400,0.9600
C01833=-21.260,114.840,29.170,-0.1000,-0.4000,0.9100
C01834=-17.710,114.630,28.880,0.0100,-0.4900,0.8700
C01835=-12.300,115.040,28.770,0.0400,-0.5100,0.8600
C01836=-6.390,115.500,28.760,0.0300,-0.5100,0.8600
C01837=0.000,115.680,28.760,0.0000,-0.5100,0.8600
C01838=0.000,114.800,30.220,0.0000,-0.5200,0.8500
C01839=-6.310,114.630,30.220,0.0300,-0.5200,0.8500
C01840=-12.170,114.170,30.220,0.0400,-0.5200,0.8500
C01841=-17.550,113.790,30.360,-0.0000,-0.5000,0.8700
C01842=-21.060,114.080,30.680,-0.1200,-0.3900,0.9100
C01843=-23.450,114.980,31.120,-0.1400,-0.2300,0.9600
C01844=-25.440,116.290,31.550,-0.0900,-0.1200,0.9900
C01845=-27.450,117.680,31.880,-0.0400,-0.0700,1.0000
C01846=-29.950,118.750,32.030,-0.0100,-0.0500,1.0000
C01847=-33.520,119.170,32.120,-0.0000,-0.0200,1.0000
C01848=-37.710,118.830,32.180,-0.0000,0.0000,1.0000
C01849=-41.900,117.720,32.250,0.0000,-0.0000,1.0000
C01850=-45.890,116.270,32.290,0.0000,-0.0000,1.0000
C01851=-49.770,114.660,32.290,0.0000,-0.0000,1.0000
C01852=-53.610,112.870,32.250,0.0000,-0.0000,1.0000
C01853=-57.360,110.690,32.180,-0.0000,0.0000,1.0000
C01854=-60.560,107.960,32.120,0.0100,-0.0100,1.0000
C01855=-62.790,105.150,32.030,0.0400,-0.0300,1.0000
C01856=-63.800,102.630,31.880,0.0800,-0.0200,1.0000
C01857=-64.240,100.220,31.550,0.1500,-0.0200,0.9900
C01858=-64.720,97.890,31.120,0.2600,-0.0600,0.9600
C01859=-65.770,95.560,30.680,0.3600,-0.2000,0.9100
C01860=-68.060,92.870,30.360,0.3500,-0.3500,0.8700
C01861=-72.130,89.340,30.220,0.3400,-0.4000,0.8500
C01862=-76.590,85.510,30.220,0.3500,-0.3900,0.8500
C01863=-81.180,81.180,30.220,0.3700,-0.3700,0.8500
C01864=-85.510,76.590,30.220,0.3900,-0.3500,0.8500
C01865=-89.340,72.130,30.220,0.4000,-0.3400,0.8500
C01866=-92.870,68.060,30.360,0.3500,-0.3500,0.8700
C01867=-95.560,65.770,30.680,0.2000,-0.3600,0.9100
C01868=-97.890,64.720,31.120,0.0600,-0.2600,0.9600
C01869=-100.220,64.240,31.550,0.0200,-0.1500,0.9900
C01870=-102.630,63.800,31.880,0.0200,-0.0800,1.0000
C01871=-105.150,62.790,32.030,0.0300,-0.0400,1.0000
C01872=-107.960,60.560,32.120,0.0100,-0.0100,1.0000
C01873=-110.690,57.360,32.180,-0.0000,0.0000,1.0000
C01874=-112.870,53.610,32.250,0.0000,-0.0000,1.0000
C01875=-114.660,49.770,32.290,0.0000,-0.0000,1.0000
C01876=-116.270,45.890,32.290,0.0000,-0.0000,1.0000
C01877=-117.720,41.900,32.250,0.0000,-0.0000,1.0000
C01878=-118.830,37.710,32.180,-0.0000,0.0000,1.0000
C01879=-119.170,33.520,32.120,0.0200,0.0000,1.0000
C01880=-118.750,29.950,32.030,0.0500,0.0100,1.0000
C01881=-117.680,27.450,31.880,0.0700,0.0400,1.0000
C01882=-116.290,25.440,31.550,0.1200,0.0900,0.9900
C01883=-114.980,23.450,31.120,0.2300,0.1400,0.9600
C01884=-114.080,21.060,30.680,0.3900,0.1200,0.9100
C01885=-113.790,17.550,30.360,0.5000,0.0000,0.8700
C01886=-114.170,12.170,30.220,0.5200,-0.0400,0.8500
C01887=-114.630,6.310,30.220,0.5200,-0.0300,0.8500
C01888=-114.800,0.000,30.220,0.5200,-0.0000,0.8500
C01889=-114.630,-6.310,30.220,0.5200,0.0300,0.8500
C01890=-114.170,-12.170,30.220,0.5200,0.0400,0.8500
C01891=-113.790,-17.540,30.360,0.5000,-0.0000,0.8700
C01892=-114.080,-21.060,30.680,0.3900,-0.1200,0.9100
C01893=-114.980,-23.450,31.120,0.2300,-0.1400,0.9600
C01894=-116.290,-25.440,31.550,0.1200,-0.0900,0.9900
C01895=-117.680,-27.450,31.880,0.0700,-0.0400,1.0000
C01896=-118.750,-29.950,32.030,0.0500,-0.0100,1.0000
C01897=-119.170,-33.520,32.120,0.0200,-0.0000,1.0000
C01898=-118.830,-37.710,32.180,-0.0000,-0.0000,1.0000
C01899=-117.720,-41.900,32.250,0.0000,0.0000,1.0000
C01900=-116.270,-45.890,32.290,0.0000,0.0000,1.0000
C01901=-114.660,-49.770,32.290,0.0000,0.0000,1.0000
C01902=-112.870,-53.610,32.250,0.0000,0.0000,1.0000
C01903=-110.690,-57.360,32.180,-0.0000,-0.0000,1.0000
C01904=-107.960,-60.560,32.120,0.0100,0.0100,1.0000
C01905=-105.150,-62.790,32.030,0.0300,0.0400,1.0000
C01906=-102.630,-63.800,31.880,0.0200,0.0800,1.0000
C01907=-100.220,-64.240,31.550,0.0200,0.1500,0.9900
C01908=-97.890,-64.720,31.120,0.0600,0.2600,0.9600
C01909=-95.560,-65.770,30.680,0.2000,0.3600,0.9100
C01910=-92.870,-68.060,30.360,0.3500,0.3500,0.8700
C01911=-89.340,-72.130,30.220,0.4000,0.3400,0.8500
C01912=-85.510,-76.590,30.220,0.3900,0.3500,0.8500
C01913=-81.180,-81.180,30.220,0.3700,0.3700,0.8500
C01914=-76.590,-85.510,30.220,0.3500,0.3900,0.8500
C01915=-72.130,-89.340,30.220,0.3400,0.4000,0.8500
C01916=-68.060,-92.870,30.360,0.3500,0.3500,0.8700
C01917=-65.770,-95.560,30.680,0.3600,0.2000,0.9100
C01918=-64.720,-97.890,31.120,0.2600,0.0600,0.9600
C01919=-64.240,-100.220,31.550,0.1500,0.0200,0.9900
C01920=-63.800,-102.630,31.880,0.0800,0.0200,1.0000
C01921=-62.790,-105.150,32.030,0.0400,0.0300,1.0000
C01922=-60.560,-107.960,32.120,0.0100,0.0100,1.0000
C01923=-57.360,-110.690,32.180,-0.0000,-0.0000,1.0000
C01924=-53.610,-112.870,32.250,0.0000,0.0000,1.0000
